RoboDK station: kr30 cnc 041719 works.rdk

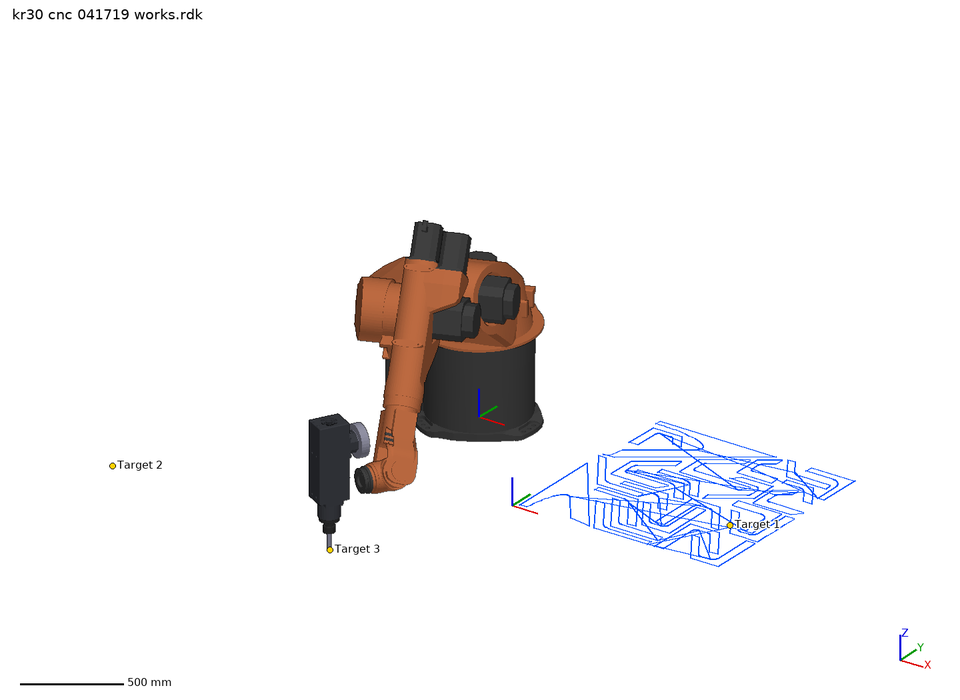
[picture v0: the station drawn from its stored meshes, robots at their saved joint values, targets as dots, program paths as lines]
Station kr30 cnc 041719 works. Poses are relative to the parent item; angles as X-Y-Z fixed-axis rotations.
  - frame KUKA KR 30 HA Base at (0, 0, 0) mm
    - robot KUKA KR 30 HA: 6 axes, payload 30 kg, reach 2033 mm, repeatability 0.05 mm, weight 665 kg
        modified DH rows (alpha deg, a mm, theta deg, d mm): 0, 0, 0, 815; -90, 350, 0, 0; 0, 850, -90, 0; -90, 145, 0, 820; 90, 0, 0, 0; -90, 0, 180, 170
        joint limits [-185, -135, -120, -350, -119, -350] to [185, 35, 158, 350, 119, 350]; home [0, -90, 90, 0, 0, 0]; saved at [68.71, -19.11, 71.06, -56.39, -66.58, 30.88]
      - tool 1/2" End Mill TCP, TCP at (337.71, -2.2, 160.57) mm, size 692.9 x 170 x 256 mm
    - frame Reference Rhino at (909.29, -1020.53, 189.15) mm
      - object RhinoPart at (0, 0, 0) mm
      - target Target 1 (Cartesian target) at (994.45, 406.4, 10) mm, rotated rx 0 ry 90 rz -60.43 deg; joints [10.582, -19.112, 71.071, -56.398, -66.586, 30.882] of KUKA KR 30 HA
      - target Target 2 (Cartesian target) at (-1810.84, -765.32, 10.08) mm, rotated rx 49.23 ry 89.99 rz -110.09 deg; joints [109.49, -19.11, 71.06, -56.39, -66.58, 30.88] of KUKA KR 30 HA
      - target Target 3 (Cartesian target) at (-425.52, -920.6, 10.08) mm, rotated rx 49.23 ry 89.99 rz -69.31 deg; joints [68.71, -19.11, 71.06, -56.39, -66.58, 30.88] of KUKA KR 30 HA
  - machining project RhinoPart Settings: C:/Users/Julian Ramirez.DESKTOP-JVDE542/Desktop/ELMER SHEET 1 TEST 3.nc | rotZ(0) | rotX(00)*rotY(360) | rotZ(0)*rotY(270)
  - object box at (500, 500, 500) mm, size 250 x 250 x 250 mm, geometry from box.sld
  - program RhinoPart (703 instructions, listed below)
  - program Prog2 (1 instructions, listed below)
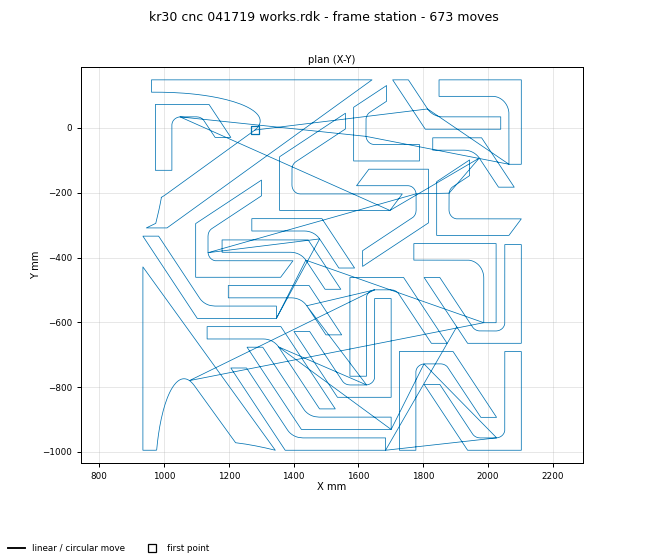
[picture p0: tool path of kr30 cnc 041719 works.rdk in frame station, 673 of 674 moves have a stored position in this frame; points joined in program order, loops and branches not executed]

--- program RhinoPart (robot KUKA KR 30 HA) ---
  Smooth(1)
  Set Ref.: Reference Rhino
  Set Tool: 1/2" End Mill TCP
  Show 1/2" End Mill TCP
  Set speed (2000.0 mm/s)
  MoveJ 1 to (371.32, 1014.09, 0) mm, rotated rx 0 ry 90 rz -60.43 deg; joints [-14.148, -38.783, 129.007, -74.576, -90.059, -0.215]
  MoveL 2 to (371.32, 1014.09, 0) mm, rotated rx 0 ry 90 rz -60.43 deg; joints [-14.148, -38.783, 129.007, -74.576, -90.059, -0.215]
  MoveL 3 to (371.32, 1014.09, 0) mm, rotated rx 0 ry 90 rz -60.43 deg; joints [-14.148, -38.783, 129.007, -74.576, -90.059, -0.215]
  Set speed (60.0 mm/s)
  MoveL 4 to (375.76, 1018.13, 0) mm, rotated rx 0 ry 90 rz -60.43 deg; joints [-14.288, -38.713, 128.612, -74.716, -89.973, 0.097]
  MoveL 5 to (379.48, 1022.21, 0) mm, rotated rx 0 ry 90 rz -60.43 deg; joints [-14.437, -38.65, 128.267, -74.866, -89.9, 0.369]
  MoveL 6 to (382.49, 1026.31, 0) mm, rotated rx 0 ry 90 rz -60.43 deg; joints [-14.595, -38.595, 127.972, -75.024, -89.839, 0.602]
  MoveL 7 to (384.79, 1030.42, 0) mm, rotated rx 0 ry 90 rz -60.43 deg; joints [-14.761, -38.548, 127.726, -75.191, -89.79, 0.795]
  MoveL 8 to (386.4, 1034.54, 0) mm, rotated rx 0 ry 90 rz -60.43 deg; joints [-14.936, -38.511, 127.53, -75.366, -89.752, 0.949]
  MoveL 9 to (387.31, 1038.67, 0) mm, rotated rx 0 ry 90 rz -60.43 deg; joints [-15.118, -38.482, 127.383, -75.549, -89.726, 1.064]
  MoveL 10 to (387.53, 1042.79, 0) mm, rotated rx 0 ry 90 rz -60.43 deg; joints [-15.309, -38.463, 127.286, -75.741, -89.71, 1.141]
  MoveL 11 to (387.07, 1046.9, 0) mm, rotated rx 0 ry 90 rz -60.43 deg; joints [-15.508, -38.454, 127.237, -75.939, -89.704, 1.18]
  MoveL 12 to (385.93, 1051, 0) mm, rotated rx 0 ry 90 rz -60.43 deg; joints [-15.715, -38.454, 127.237, -76.146, -89.709, 1.181]
  MoveL 13 to (384.11, 1055.07, 0) mm, rotated rx 0 ry 90 rz -60.43 deg; joints [-15.929, -38.463, 127.285, -76.36, -89.722, 1.145]
  MoveL 14 to (381.63, 1059.1, 0) mm, rotated rx 0 ry 90 rz -60.43 deg; joints [-16.152, -38.482, 127.38, -76.582, -89.744, 1.071]
  MoveL 15 to (378.49, 1063.11, 0) mm, rotated rx 0 ry 90 rz -60.43 deg; joints [-16.382, -38.509, 127.523, -76.812, -89.775, 0.96]
  MoveL 16 to (374.68, 1067.06, 0) mm, rotated rx 0 ry 90 rz -60.43 deg; joints [-16.62, -38.546, 127.713, -77.05, -89.813, 0.812]
  MoveL 17 to (370.23, 1070.97, 0) mm, rotated rx 0 ry 90 rz -60.43 deg; joints [-16.866, -38.59, 127.949, -77.295, -89.859, 0.626]
  MoveL 18 to (365.13, 1074.81, 0) mm, rotated rx 0 ry 90 rz -60.43 deg; joints [-17.12, -38.643, 128.23, -77.548, -89.911, 0.403]
  MoveL 19 to (356.11, 1080.56, 0) mm, rotated rx 0 ry 90 rz -60.43 deg; joints [-17.523, -38.737, 128.745, -77.951, -90.002, -0.008]
  MoveL 20 to (346.45, 1085.73, 0) mm, rotated rx 0 ry 90 rz -60.43 deg; joints [-17.913, -38.837, 129.313, -78.342, -90.096, -0.467]
  MoveL 21 to (336.49, 1090.32, 0) mm, rotated rx 0 ry 90 rz -60.43 deg; joints [-18.286, -38.938, 129.909, -78.716, -90.19, -0.953]
  MoveL 22 to (326.6, 1094.34, 0) mm, rotated rx 0 ry 90 rz -60.43 deg; joints [-18.636, -39.034, 130.507, -79.068, -90.279, -1.446]
  MoveL 23 to (304.84, 1101.8, 0) mm, rotated rx 0 ry 90 rz -60.43 deg; joints [-19.356, -39.233, 131.838, -79.794, -90.462, -2.563]
  MoveL 24 to (282.07, 1108.12, 0) mm, rotated rx 0 ry 90 rz -60.43 deg; joints [-20.061, -39.416, 133.239, -80.511, -90.631, -3.77]
  MoveL 25 to (259.04, 1113.38, 0) mm, rotated rx 0 ry 90 rz -60.43 deg; joints [-20.745, -39.572, 134.659, -81.207, -90.78, -5.027]
  MoveL 26 to (236.49, 1117.66, 0) mm, rotated rx 0 ry 90 rz -60.43 deg; joints [-21.394, -39.693, 136.047, -81.872, -90.902, -6.29]
  MoveL 27 to (215.72, 1120.95, 0) mm, rotated rx 0 ry 90 rz -60.43 deg; joints [-21.981, -39.774, 137.321, -82.474, -90.994, -7.481]
  MoveL 28 to (194.75, 1123.72, 0) mm, rotated rx 0 ry 90 rz -60.43 deg; joints [-22.566, -39.826, 138.602, -83.075, -91.066, -8.712]
  MoveL 29 to (173.72, 1126.01, 0) mm, rotated rx 0 ry 90 rz -60.43 deg; joints [-23.147, -39.843, 139.881, -83.673, -91.117, -9.976]
  MoveL 30 to (152.78, 1127.82, 0) mm, rotated rx 0 ry 90 rz -60.43 deg; joints [-23.724, -39.824, 141.147, -84.265, -91.146, -11.265]
  MoveL 31 to (132.99, 1129.14, 0) mm, rotated rx 0 ry 90 rz -60.43 deg; joints [-24.268, -39.771, 142.336, -84.822, -91.152, -12.513]
  MoveL 32 to (116.9, 1129.95, 0) mm, rotated rx 0 ry 90 rz -60.43 deg; joints [-24.71, -39.701, 143.298, -85.274, -91.142, -13.55]
  MoveL 33 to (100.77, 1130.52, 0) mm, rotated rx 0 ry 90 rz -60.43 deg; joints [-25.154, -39.606, 144.257, -85.725, -91.116, -14.609]
  MoveL 34 to (84.64, 1130.87, 0) mm, rotated rx 0 ry 90 rz -60.43 deg; joints [-25.598, -39.482, 145.211, -86.175, -91.076, -15.692]
  MoveL 35 to (68.52, 1130.98, 0) mm, rotated rx 0 ry 90 rz -60.43 deg; joints [-26.044, -39.331, 146.159, -86.623, -91.021, -16.798]
  MoveL 36 to (51.93, 1130.98, 0) mm, rotated rx 0 ry 90 rz -60.43 deg; joints [-26.511, -39.143, 147.126, -87.088, -90.945, -17.959]
  MoveL 37 to (51.93, 1169.08, 0) mm, rotated rx 0 ry 90 rz -60.43 deg; joints [-28.654, -39.362, 145.978, -89.121, -90.262, -16.614]
  MoveL 38 to (732.85, 1169.08, 0) mm, rotated rx 0 ry 90 rz -60.43 deg; joints [-16.446, -29.001, 96.264, -77.863, -84.965, 22.201]
  MoveL 39 to (99.83, 711.88, 0) mm, rotated rx 0 ry 90 rz -60.43 deg; joints [1.355, -38.347, 150.049, -60.898, -100.955, -18.85]
  MoveL 40 to (36.02, 711.88, 0) mm, rotated rx 0 ry 90 rz -60.43 deg; joints [1.465, -36.599, 153.958, -61.879, -103.707, -23.912]
  MoveL 41 to (65.11, 725.98, 0) mm, rotated rx 0 ry 90 rz -60.43 deg; joints [0.419, -37.491, 152.214, -62.335, -102.067, -21.741]
  MoveL 42 to (69.92, 745.6, 0) mm, rotated rx 0 ry 90 rz -60.43 deg; joints [-0.957, -37.626, 151.913, -63.561, -101.361, -21.61]
  MoveL 43 to (74.45, 765.38, 0) mm, rotated rx 0 ry 90 rz -60.43 deg; joints [-2.329, -37.76, 151.6, -64.782, -100.662, -21.448]
  MoveL 44 to (78.62, 785.23, 0) mm, rotated rx 0 ry 90 rz -60.43 deg; joints [-3.689, -37.892, 151.279, -65.995, -99.978, -21.26]
  MoveL 45 to (82.38, 805.12, 0) mm, rotated rx 0 ry 90 rz -60.43 deg; joints [-5.036, -38.021, 150.952, -67.198, -99.311, -21.05]
  MoveL 46 to (81.84, 806.04, 0) mm, rotated rx 0 ry 90 rz -60.43 deg; joints [-5.103, -38.01, 150.981, -67.267, -99.302, -21.097]
  MoveL 47 to (85.5, 808.13, 0) mm, rotated rx 0 ry 90 rz -60.43 deg; joints [-5.223, -38.1, 150.742, -67.332, -99.132, -20.808]
  MoveL 48 to (89.1, 810.32, 0) mm, rotated rx 0 ry 90 rz -60.43 deg; joints [-5.349, -38.187, 150.506, -67.404, -98.964, -20.525]
  MoveL 49 to (92.62, 812.61, 0) mm, rotated rx 0 ry 90 rz -60.43 deg; joints [-5.481, -38.27, 150.274, -67.484, -98.797, -20.25]
  MoveL 50 to (96.07, 815.01, 0) mm, rotated rx 0 ry 90 rz -60.43 deg; joints [-5.621, -38.349, 150.044, -67.572, -98.631, -19.981]
  MoveL 51 to (366.16, 1010.08, 0) mm, rotated rx 0 ry 90 rz -60.43 deg; joints [-14.016, -38.861, 129.451, -74.446, -90.158, -0.569]
  MoveL 52 to (371.32, 1014.09, 0) mm, rotated rx 0 ry 90 rz -60.43 deg; joints [-14.148, -38.783, 129.007, -74.576, -90.059, -0.215]
  MoveL 53 to (904.53, 1079.22, 0) mm, rotated rx 0 ry 90 rz -60.43 deg; joints [-11.868, -22.969, 81.101, -74.832, -80.761, 30.636]
  Set speed (60.0 mm/s)
  MoveL 54 to (845.14, 1169.08, 0) mm, rotated rx 0 ry 90 rz -60.43 deg; joints [-15.343, -24.65, 85.19, -77.55, -83.057, 28.702]
  MoveL 55 to (796.61, 1169.08, 0) mm, rotated rx 0 ry 90 rz -60.43 deg; joints [-15.802, -26.637, 90.145, -77.629, -83.905, 25.83]
  MoveL 56 to (897.33, 1016.68, 0) mm, rotated rx 0 ry 90 rz -60.43 deg; joints [-9.818, -23.849, 83.23, -72.827, -80.088, 29.119]
  MoveL 57 to (1130.3, 1016.68, 0) mm, rotated rx 0 ry 90 rz -60.43 deg; joints [-8.62, -9.728, 50.987, -75.829, -74.407, 46.791]
  MoveL 58 to (1130.3, 1054.78, 0) mm, rotated rx 0 ry 90 rz -60.43 deg; joints [-9.753, -9.185, 49.806, -76.795, -75.087, 47.643]
  MoveL 59 to (951.82, 1054.78, 0) mm, rotated rx 0 ry 90 rz -60.43 deg; joints [-10.754, -20.904, 76.185, -74.352, -79.414, 33.26]
  MoveL 60 to (948.36, 1054.88, 0) mm, rotated rx 0 ry 90 rz -60.43 deg; joints [-10.778, -21.079, 76.597, -74.331, -79.491, 33.032]
  MoveL 61 to (944.91, 1055.18, 0) mm, rotated rx 0 ry 90 rz -60.43 deg; joints [-10.81, -21.25, 77, -74.316, -79.571, 32.809]
  MoveL 62 to (941.49, 1055.67, 0) mm, rotated rx 0 ry 90 rz -60.43 deg; joints [-10.847, -21.416, 77.394, -74.308, -79.653, 32.592]
  MoveL 63 to (938.11, 1056.36, 0) mm, rotated rx 0 ry 90 rz -60.43 deg; joints [-10.891, -21.578, 77.777, -74.307, -79.736, 32.383]
  MoveL 64 to (934.77, 1057.25, 0) mm, rotated rx 0 ry 90 rz -60.43 deg; joints [-10.941, -21.734, 78.148, -74.313, -79.821, 32.181]
  MoveL 65 to (931.48, 1058.34, 0) mm, rotated rx 0 ry 90 rz -60.43 deg; joints [-10.998, -21.885, 78.506, -74.326, -79.907, 31.986]
  MoveL 66 to (928.27, 1059.61, 0) mm, rotated rx 0 ry 90 rz -60.43 deg; joints [-11.06, -22.029, 78.85, -74.346, -79.994, 31.801]
  MoveL 67 to (925.13, 1061.08, 0) mm, rotated rx 0 ry 90 rz -60.43 deg; joints [-11.129, -22.167, 79.179, -74.373, -80.082, 31.624]
  MoveL 68 to (922.08, 1062.74, 0) mm, rotated rx 0 ry 90 rz -60.43 deg; joints [-11.204, -22.298, 79.492, -74.407, -80.17, 31.457]
  MoveL 69 to (919.14, 1064.59, 0) mm, rotated rx 0 ry 90 rz -60.43 deg; joints [-11.284, -22.422, 79.786, -74.448, -80.258, 31.302]
  MoveL 70 to (916.32, 1066.61, 0) mm, rotated rx 0 ry 90 rz -60.43 deg; joints [-11.37, -22.536, 80.061, -74.496, -80.345, 31.158]
  MoveL 71 to (913.65, 1068.81, 0) mm, rotated rx 0 ry 90 rz -60.43 deg; joints [-11.46, -22.642, 80.315, -74.551, -80.431, 31.026]
  MoveL 72 to (911.12, 1071.17, 0) mm, rotated rx 0 ry 90 rz -60.43 deg; joints [-11.556, -22.739, 80.547, -74.612, -80.516, 30.908]
  MoveL 73 to (908.75, 1073.7, 0) mm, rotated rx 0 ry 90 rz -60.43 deg; joints [-11.656, -22.826, 80.756, -74.679, -80.599, 30.803]
  MoveL 74 to (906.55, 1076.38, 0) mm, rotated rx 0 ry 90 rz -60.43 deg; joints [-11.76, -22.903, 80.941, -74.752, -80.681, 30.712]
  MoveL 75 to (904.53, 1079.22, 0) mm, rotated rx 0 ry 90 rz -60.43 deg; joints [-11.868, -22.969, 81.101, -74.832, -80.761, 30.636]
  MoveL 76 to (1155.7, 908.41, 0) mm, rotated rx 0 ry 90 rz -60.43 deg; joints [-5.296, -8.63, 48.604, -73.841, -71.636, 47.397]
  Set speed (60.0 mm/s)
  MoveL 77 to (1155.7, 1062.81, 0) mm, rotated rx 0 ry 90 rz -60.43 deg; joints [-9.86, -6.6, 44.232, -77.66, -74.507, 50.684]
  MoveL 78 to (1155.47, 1068.04, 0) mm, rotated rx 0 ry 90 rz -60.43 deg; joints [-10.014, -6.528, 44.077, -77.784, -74.609, 50.794]
  MoveL 79 to (1154.79, 1073.23, 0) mm, rotated rx 0 ry 90 rz -60.43 deg; joints [-10.169, -6.503, 44.023, -77.893, -74.723, 50.85]
  MoveL 80 to (1153.66, 1078.33, 0) mm, rotated rx 0 ry 90 rz -60.43 deg; joints [-10.323, -6.525, 44.07, -77.987, -74.848, 50.852]
  MoveL 81 to (1152.09, 1083.3, 0) mm, rotated rx 0 ry 90 rz -60.43 deg; joints [-10.477, -6.594, 44.218, -78.067, -74.983, 50.797]
  MoveL 82 to (1150.07, 1088.11, 0) mm, rotated rx 0 ry 90 rz -60.43 deg; joints [-10.628, -6.71, 44.467, -78.131, -75.128, 50.688]
  MoveL 83 to (1147.63, 1092.73, 0) mm, rotated rx 0 ry 90 rz -60.43 deg; joints [-10.776, -6.872, 44.815, -78.18, -75.28, 50.525]
  MoveL 84 to (1144.76, 1097.1, 0) mm, rotated rx 0 ry 90 rz -60.43 deg; joints [-10.919, -7.079, 45.259, -78.214, -75.44, 50.309]
  MoveL 85 to (1141.47, 1101.2, 0) mm, rotated rx 0 ry 90 rz -60.43 deg; joints [-11.058, -7.329, 45.797, -78.233, -75.605, 50.041]
  MoveL 86 to (1137.81, 1104.95, 0) mm, rotated rx 0 ry 90 rz -60.43 deg; joints [-11.189, -7.618, 46.419, -78.237, -75.772, 49.726]
  MoveL 87 to (1133.82, 1108.29, 0) mm, rotated rx 0 ry 90 rz -60.43 deg; joints [-11.309, -7.94, 47.112, -78.226, -75.94, 49.37]
  MoveL 88 to (1129.54, 1111.18, 0) mm, rotated rx 0 ry 90 rz -60.43 deg; joints [-11.419, -8.29, 47.868, -78.201, -76.106, 48.979]
  MoveL 89 to (1125, 1113.61, 0) mm, rotated rx 0 ry 90 rz -60.43 deg; joints [-11.518, -8.664, 48.679, -78.163, -76.269, 48.556]
  MoveL 90 to (1120.24, 1115.55, 0) mm, rotated rx 0 ry 90 rz -60.43 deg; joints [-11.603, -9.06, 49.536, -78.112, -76.428, 48.105]
  MoveL 91 to (1115.28, 1116.96, 0) mm, rotated rx 0 ry 90 rz -60.43 deg; joints [-11.675, -9.473, 50.432, -78.048, -76.581, 47.63]
  MoveL 92 to (1110.15, 1117.83, 0) mm, rotated rx 0 ry 90 rz -60.43 deg; joints [-11.732, -9.899, 51.36, -77.971, -76.727, 47.134]
  MoveL 93 to (1104.9, 1118.13, 0) mm, rotated rx 0 ry 90 rz -60.43 deg; joints [-11.773, -10.337, 52.314, -77.881, -76.865, 46.622]
  MoveL 94 to (939.8, 1118.13, 0) mm, rotated rx 0 ry 90 rz -60.43 deg; joints [-12.888, -20.841, 76.037, -76.175, -80.569, 33.658]
  MoveL 95 to (939.8, 1169.08, 0) mm, rotated rx 0 ry 90 rz -60.43 deg; joints [-14.52, -20.204, 74.544, -77.675, -81.292, 34.719]
  MoveL 96 to (1193.8, 1169.08, 0) mm, rotated rx 0 ry 90 rz -60.43 deg; joints [-12.687, 1.86, 26.402, -81.821, -75.178, 60.673]
  MoveL 97 to (1193.8, 908.41, 0) mm, rotated rx 0 ry 90 rz -60.43 deg; joints [-5.193, -4.605, 39.971, -75.302, -70.33, 52.072]
  MoveL 98 to (1155.7, 908.41, 0) mm, rotated rx 0 ry 90 rz -60.43 deg; joints [-5.296, -8.63, 48.604, -73.841, -71.636, 47.397]
  MoveL 99 to (714.35, 994.58, 0) mm, rotated rx 0 ry 90 rz -60.43 deg; joints [-10.182, -31.026, 101.761, -71.621, -83.712, 18.246]
  Set speed (60.0 mm/s)
  MoveL 100 to (714.24, 997.2, 0) mm, rotated rx 0 ry 90 rz -60.43 deg; joints [-10.282, -31.014, 101.729, -71.719, -83.736, 18.276]
  MoveL 101 to (714.24, 1045.45, 0) mm, rotated rx 0 ry 90 rz -60.43 deg; joints [-12.101, -30.702, 100.864, -73.508, -84.152, 18.99]
  MoveL 102 to (714.44, 1048.91, 0) mm, rotated rx 0 ry 90 rz -60.43 deg; joints [-12.229, -30.671, 100.778, -73.635, -84.179, 19.055]
  MoveL 103 to (715.04, 1052.32, 0) mm, rotated rx 0 ry 90 rz -60.43 deg; joints [-12.352, -30.627, 100.656, -73.76, -84.197, 19.142]
  MoveL 104 to (716.03, 1055.63, 0) mm, rotated rx 0 ry 90 rz -60.43 deg; joints [-12.467, -30.57, 100.5, -73.879, -84.207, 19.249]
  MoveL 105 to (717.39, 1058.8, 0) mm, rotated rx 0 ry 90 rz -60.43 deg; joints [-12.574, -30.502, 100.312, -73.992, -84.209, 19.375]
  MoveL 106 to (719.13, 1061.77, 0) mm, rotated rx 0 ry 90 rz -60.43 deg; joints [-12.67, -30.422, 100.094, -74.096, -84.203, 19.518]
  MoveL 107 to (721.23, 1064.5, 0) mm, rotated rx 0 ry 90 rz -60.43 deg; joints [-12.754, -30.332, 99.846, -74.191, -84.188, 19.678]
  MoveL 108 to (723.67, 1066.96, 0) mm, rotated rx 0 ry 90 rz -60.43 deg; joints [-12.824, -30.231, 99.571, -74.275, -84.165, 19.853]
  MoveL 109 to (726.46, 1069.09, 0) mm, rotated rx 0 ry 90 rz -60.43 deg; joints [-12.88, -30.121, 99.271, -74.346, -84.132, 20.043]
  MoveL 110 to (777.74, 1102.98, 0) mm, rotated rx 0 ry 90 rz -60.43 deg; joints [-13.668, -28.021, 93.695, -75.446, -83.519, 23.498]
  MoveL 111 to (777.74, 1151.51, 0) mm, rotated rx 0 ry 90 rz -60.43 deg; joints [-15.376, -27.55, 92.477, -77.095, -84.035, 24.398]
  MoveL 112 to (676.14, 1084.36, 0) mm, rotated rx 0 ry 90 rz -60.43 deg; joints [-13.899, -31.631, 103.464, -75.073, -85.169, 17.533]
  MoveL 113 to (676.14, 918.58, 0) mm, rotated rx 0 ry 90 rz -60.43 deg; joints [-7.466, -32.586, 106.219, -68.709, -83.913, 15.221]
  MoveL 114 to (879.34, 918.58, 0) mm, rotated rx 0 ry 90 rz -60.43 deg; joints [-6.543, -25.264, 86.704, -69.527, -79.221, 26.607]
  MoveL 115 to (879.34, 969.54, 0) mm, rotated rx 0 ry 90 rz -60.43 deg; joints [-8.307, -24.977, 85.996, -71.199, -79.879, 27.302]
  MoveL 116 to (739.64, 969.54, 0) mm, rotated rx 0 ry 90 rz -60.43 deg; joints [-9.074, -30.328, 99.837, -70.701, -82.959, 19.293]
  MoveL 117 to (737.01, 969.69, 0) mm, rotated rx 0 ry 90 rz -60.43 deg; joints [-9.096, -30.416, 100.077, -70.704, -83.016, 19.151]
  MoveL 118 to (734.45, 970.12, 0) mm, rotated rx 0 ry 90 rz -60.43 deg; joints [-9.127, -30.5, 100.307, -70.717, -83.075, 19.015]
  MoveL 119 to (731.97, 970.83, 0) mm, rotated rx 0 ry 90 rz -60.43 deg; joints [-9.169, -30.579, 100.524, -70.741, -83.134, 18.889]
  MoveL 120 to (729.59, 971.8, 0) mm, rotated rx 0 ry 90 rz -60.43 deg; joints [-9.22, -30.653, 100.728, -70.775, -83.193, 18.771]
  MoveL 121 to (727.32, 973.01, 0) mm, rotated rx 0 ry 90 rz -60.43 deg; joints [-9.28, -30.722, 100.918, -70.819, -83.252, 18.662]
  MoveL 122 to (725.18, 974.46, 0) mm, rotated rx 0 ry 90 rz -60.43 deg; joints [-9.348, -30.785, 101.092, -70.871, -83.311, 18.564]
  MoveL 123 to (723.19, 976.13, 0) mm, rotated rx 0 ry 90 rz -60.43 deg; joints [-9.424, -30.841, 101.249, -70.932, -83.367, 18.477]
  MoveL 124 to (721.35, 978, 0) mm, rotated rx 0 ry 90 rz -60.43 deg; joints [-9.507, -30.891, 101.387, -71.002, -83.422, 18.402]
  MoveL 125 to (719.71, 980.05, 0) mm, rotated rx 0 ry 90 rz -60.43 deg; joints [-9.595, -30.934, 101.505, -71.078, -83.475, 18.34]
  MoveL 126 to (718.27, 982.24, 0) mm, rotated rx 0 ry 90 rz -60.43 deg; joints [-9.687, -30.968, 101.602, -71.159, -83.524, 18.291]
  MoveL 127 to (717.05, 984.54, 0) mm, rotated rx 0 ry 90 rz -60.43 deg; joints [-9.783, -30.995, 101.677, -71.245, -83.569, 18.255]
  MoveL 128 to (716.05, 986.95, 0) mm, rotated rx 0 ry 90 rz -60.43 deg; joints [-9.881, -31.015, 101.73, -71.335, -83.611, 18.233]
  MoveL 129 to (715.26, 989.44, 0) mm, rotated rx 0 ry 90 rz -60.43 deg; joints [-9.98, -31.026, 101.762, -71.428, -83.649, 18.224]
  MoveL 130 to (714.69, 991.99, 0) mm, rotated rx 0 ry 90 rz -60.43 deg; joints [-10.081, -31.03, 101.773, -71.524, -83.682, 18.229]
  MoveL 131 to (714.35, 994.58, 0) mm, rotated rx 0 ry 90 rz -60.43 deg; joints [-10.182, -31.026, 101.761, -71.621, -83.712, 18.246]
  MoveL 132 to (139.93, 1054.78, 0) mm, rotated rx 0 ry 90 rz -60.43 deg; joints [-19.98, -39.656, 143.784, -80.693, -92.331, -13.939]
  Set speed (60.0 mm/s)
  MoveL 133 to (137.34, 1054.44, 0) mm, rotated rx 0 ry 90 rz -60.43 deg; joints [-20.014, -39.639, 143.955, -80.734, -92.353, -14.125]
  MoveL 134 to (134.79, 1053.88, 0) mm, rotated rx 0 ry 90 rz -60.43 deg; joints [-20.035, -39.62, 144.127, -80.762, -92.378, -14.314]
  MoveL 135 to (132.3, 1053.09, 0) mm, rotated rx 0 ry 90 rz -60.43 deg; joints [-20.042, -39.601, 144.3, -80.777, -92.408, -14.505]
  MoveL 136 to (129.9, 1052.08, 0) mm, rotated rx 0 ry 90 rz -60.43 deg; joints [-20.035, -39.58, 144.473, -80.778, -92.44, -14.695]
  MoveL 137 to (127.59, 1050.86, 0) mm, rotated rx 0 ry 90 rz -60.43 deg; joints [-20.013, -39.559, 144.644, -80.765, -92.477, -14.885]
  MoveL 138 to (125.4, 1049.43, 0) mm, rotated rx 0 ry 90 rz -60.43 deg; joints [-19.976, -39.537, 144.812, -80.737, -92.517, -15.071]
  MoveL 139 to (123.35, 1047.78, 0) mm, rotated rx 0 ry 90 rz -60.43 deg; joints [-19.923, -39.515, 144.976, -80.695, -92.561, -15.253]
  MoveL 140 to (121.48, 1045.95, 0) mm, rotated rx 0 ry 90 rz -60.43 deg; joints [-19.856, -39.493, 145.134, -80.638, -92.608, -15.427]
  MoveL 141 to (119.81, 1043.95, 0) mm, rotated rx 0 ry 90 rz -60.43 deg; joints [-19.775, -39.472, 145.282, -80.567, -92.657, -15.59]
  MoveL 142 to (118.36, 1041.82, 0) mm, rotated rx 0 ry 90 rz -60.43 deg; joints [-19.68, -39.452, 145.419, -80.483, -92.709, -15.741]
  MoveL 143 to (117.15, 1039.55, 0) mm, rotated rx 0 ry 90 rz -60.43 deg; joints [-19.572, -39.433, 145.544, -80.386, -92.762, -15.879]
  MoveL 144 to (116.18, 1037.16, 0) mm, rotated rx 0 ry 90 rz -60.43 deg; joints [-19.452, -39.415, 145.656, -80.277, -92.817, -16.001]
  MoveL 145 to (115.47, 1034.68, 0) mm, rotated rx 0 ry 90 rz -60.43 deg; joints [-19.321, -39.399, 145.754, -80.155, -92.872, -16.107]
  MoveL 146 to (115.04, 1032.12, 0) mm, rotated rx 0 ry 90 rz -60.43 deg; joints [-19.178, -39.386, 145.836, -80.023, -92.928, -16.194]
  MoveL 147 to (114.89, 1029.5, 0) mm, rotated rx 0 ry 90 rz -60.43 deg; joints [-19.025, -39.375, 145.901, -79.88, -92.984, -16.262]
  MoveL 148 to (114.89, 889.8, 0) mm, rotated rx 0 ry 90 rz -60.43 deg; joints [-10.367, -38.892, 148.202, -71.802, -96.244, -18.308]
  MoveL 149 to (63.94, 889.8, 0) mm, rotated rx 0 ry 90 rz -60.43 deg; joints [-11.002, -37.862, 151.353, -72.876, -97.292, -22.391]
  MoveL 150 to (63.94, 1093, 0) mm, rotated rx 0 ry 90 rz -60.43 deg; joints [-23.973, -39.068, 147.471, -84.686, -91.765, -18.321]
  MoveL 151 to (229.71, 1093, 0) mm, rotated rx 0 ry 90 rz -60.43 deg; joints [-20.268, -39.763, 137.112, -80.771, -91.185, -7.253]
  MoveL 152 to (296.86, 991.4, 0) mm, rotated rx 0 ry 90 rz -60.43 deg; joints [-13.945, -39.574, 134.678, -74.432, -91.373, -4.916]
  MoveL 153 to (248.33, 991.4, 0) mm, rotated rx 0 ry 90 rz -60.43 deg; joints [-14.596, -39.806, 138, -75.17, -92.111, -7.92]
  MoveL 154 to (214.44, 1042.68, 0) mm, rotated rx 0 ry 90 rz -60.43 deg; joints [-17.893, -39.839, 139.265, -78.474, -91.9, -9.234]
  MoveL 155 to (212.31, 1045.46, 0) mm, rotated rx 0 ry 90 rz -60.43 deg; joints [-18.08, -39.84, 139.345, -78.662, -91.885, -9.318]
  MoveL 156 to (209.86, 1047.91, 0) mm, rotated rx 0 ry 90 rz -60.43 deg; joints [-18.256, -39.841, 139.454, -78.839, -91.878, -9.429]
  MoveL 157 to (207.12, 1050.01, 0) mm, rotated rx 0 ry 90 rz -60.43 deg; joints [-18.418, -39.842, 139.587, -79.003, -91.876, -9.564]
  MoveL 158 to (204.15, 1051.74, 0) mm, rotated rx 0 ry 90 rz -60.43 deg; joints [-18.565, -39.843, 139.744, -79.154, -91.881, -9.722]
  MoveL 159 to (200.98, 1053.11, 0) mm, rotated rx 0 ry 90 rz -60.43 deg; joints [-18.697, -39.843, 139.92, -79.289, -91.892, -9.899]
  MoveL 160 to (197.68, 1054.09, 0) mm, rotated rx 0 ry 90 rz -60.43 deg; joints [-18.811, -39.842, 140.113, -79.408, -91.908, -10.094]
  MoveL 161 to (190.8, 1054.9, 0) mm, rotated rx 0 ry 90 rz -60.43 deg; joints [-18.983, -39.838, 140.542, -79.592, -91.956, -10.526]
  MoveL 162 to (142.55, 1054.9, 0) mm, rotated rx 0 ry 90 rz -60.43 deg; joints [-19.932, -39.672, 143.618, -80.64, -92.313, -13.756]
  MoveL 163 to (139.93, 1054.78, 0) mm, rotated rx 0 ry 90 rz -60.43 deg; joints [-19.98, -39.656, 143.784, -80.693, -92.331, -13.939]
  MoveL 164 to (788.26, 765.88, 0) mm, rotated rx 0 ry 90 rz -60.43 deg; joints [-1.266, -29.269, 96.976, -63.512, -79.638, 19.847]
  Set speed (60.0 mm/s)
  MoveL 165 to (826.36, 816.83, 0) mm, rotated rx 0 ry 90 rz -60.43 deg; joints [-3.087, -27.773, 93.052, -65.649, -79.251, 22.395]
  MoveL 166 to (511.04, 816.83, 0) mm, rotated rx 0 ry 90 rz -60.43 deg; joints [-3.857, -36.982, 120.764, -64.418, -87.306, 5.606]
  MoveL 167 to (505.85, 817.41, 0) mm, rotated rx 0 ry 90 rz -60.43 deg; joints [-3.9, -37.085, 121.169, -64.448, -87.441, 5.336]
  MoveL 168 to (503.37, 818.12, 0) mm, rotated rx 0 ry 90 rz -60.43 deg; joints [-3.94, -37.133, 121.36, -64.482, -87.506, 5.208]
  MoveL 169 to (500.99, 819.09, 0) mm, rotated rx 0 ry 90 rz -60.43 deg; joints [-3.991, -37.178, 121.541, -64.528, -87.569, 5.088]
  MoveL 170 to (498.72, 820.3, 0) mm, rotated rx 0 ry 90 rz -60.43 deg; joints [-4.054, -37.221, 121.712, -64.586, -87.63, 4.974]
  MoveL 171 to (496.58, 821.75, 0) mm, rotated rx 0 ry 90 rz -60.43 deg; joints [-4.127, -37.26, 121.871, -64.654, -87.688, 4.869]
  MoveL 172 to (494.59, 823.42, 0) mm, rotated rx 0 ry 90 rz -60.43 deg; joints [-4.211, -37.296, 122.017, -64.733, -87.742, 4.772]
  MoveL 173 to (492.75, 825.29, 0) mm, rotated rx 0 ry 90 rz -60.43 deg; joints [-4.303, -37.328, 122.149, -64.822, -87.792, 4.686]
  MoveL 174 to (491.11, 827.34, 0) mm, rotated rx 0 ry 90 rz -60.43 deg; joints [-4.403, -37.357, 122.265, -64.918, -87.837, 4.61]
  MoveL 175 to (489.67, 829.53, 0) mm, rotated rx 0 ry 90 rz -60.43 deg; joints [-4.509, -37.381, 122.364, -65.021, -87.877, 4.547]
  MoveL 176 to (487.45, 834.24, 0) mm, rotated rx 0 ry 90 rz -60.43 deg; joints [-4.734, -37.415, 122.507, -65.242, -87.94, 4.456]
  MoveL 177 to (486.09, 839.28, 0) mm, rotated rx 0 ry 90 rz -60.43 deg; joints [-4.971, -37.433, 122.579, -65.477, -87.982, 4.415]
  MoveL 178 to (485.64, 844.49, 0) mm, rotated rx 0 ry 90 rz -60.43 deg; joints [-5.213, -37.432, 122.578, -65.719, -88, 4.424]
  MoveL 179 to (485.64, 892.74, 0) mm, rotated rx 0 ry 90 rz -60.43 deg; joints [-7.426, -37.332, 122.164, -67.936, -88.054, 4.789]
  MoveL 180 to (485.84, 896.21, 0) mm, rotated rx 0 ry 90 rz -60.43 deg; joints [-7.583, -37.319, 122.113, -68.094, -88.053, 4.83]
  MoveL 181 to (486.44, 899.62, 0) mm, rotated rx 0 ry 90 rz -60.43 deg; joints [-7.735, -37.299, 122.031, -68.247, -88.043, 4.892]
  MoveL 182 to (487.43, 902.93, 0) mm, rotated rx 0 ry 90 rz -60.43 deg; joints [-7.88, -37.272, 121.919, -68.394, -88.024, 4.976]
  MoveL 183 to (488.79, 906.09, 0) mm, rotated rx 0 ry 90 rz -60.43 deg; joints [-8.015, -37.237, 121.779, -68.532, -87.997, 5.079]
  MoveL 184 to (490.53, 909.06, 0) mm, rotated rx 0 ry 90 rz -60.43 deg; joints [-8.139, -37.196, 121.611, -68.66, -87.962, 5.2]
  MoveL 185 to (492.63, 911.8, 0) mm, rotated rx 0 ry 90 rz -60.43 deg; joints [-8.249, -37.148, 121.418, -68.774, -87.92, 5.34]
  MoveL 186 to (495.07, 914.25, 0) mm, rotated rx 0 ry 90 rz -60.43 deg; joints [-8.344, -37.093, 121.2, -68.874, -87.87, 5.496]
  MoveL 187 to (497.86, 916.38, 0) mm, rotated rx 0 ry 90 rz -60.43 deg; joints [-8.421, -37.032, 120.958, -68.958, -87.812, 5.667]
  MoveL 188 to (650.74, 1017.42, 0) mm, rotated rx 0 ry 90 rz -60.43 deg; joints [-11.535, -32.847, 106.99, -72.608, -85.147, 15.114]
  MoveL 189 to (650.74, 1065.95, 0) mm, rotated rx 0 ry 90 rz -60.43 deg; joints [-13.43, -32.533, 106.064, -74.488, -85.48, 15.852]
  MoveL 190 to (447.54, 931.66, 0) mm, rotated rx 0 ry 90 rz -60.43 deg; joints [-9.484, -37.91, 124.64, -69.942, -88.877, 3.071]
  MoveL 191 to (447.54, 765.88, 0) mm, rotated rx 0 ry 90 rz -60.43 deg; joints [-1.626, -38.176, 125.869, -62.074, -88.919, 2.038]
  MoveL 192 to (788.26, 765.88, 0) mm, rotated rx 0 ry 90 rz -60.43 deg; joints [-1.266, -29.269, 96.976, -63.512, -79.638, 19.847]
  MoveL 193 to (1064.06, 927.56, 0) mm, rotated rx 0 ry 90 rz -60.43 deg; joints [-6.162, -15.538, 63.842, -72.085, -74.676, 39.266]
  Set speed (60.0 mm/s)
  MoveL 194 to (1062.04, 930.4, 0) mm, rotated rx 0 ry 90 rz -60.43 deg; joints [-6.257, -15.649, 64.092, -72.126, -74.779, 39.149]
  MoveL 195 to (1059.84, 933.08, 0) mm, rotated rx 0 ry 90 rz -60.43 deg; joints [-6.349, -15.772, 64.37, -72.16, -74.884, 39.016]
  MoveL 196 to (1057.47, 935.61, 0) mm, rotated rx 0 ry 90 rz -60.43 deg; joints [-6.436, -15.906, 64.673, -72.187, -74.991, 38.868]
  MoveL 197 to (1054.94, 937.97, 0) mm, rotated rx 0 ry 90 rz -60.43 deg; joints [-6.519, -16.051, 64.999, -72.208, -75.098, 38.706]
  MoveL 198 to (1052.26, 940.17, 0) mm, rotated rx 0 ry 90 rz -60.43 deg; joints [-6.598, -16.204, 65.347, -72.222, -75.207, 38.531]
  MoveL 199 to (1049.45, 942.19, 0) mm, rotated rx 0 ry 90 rz -60.43 deg; joints [-6.672, -16.367, 65.715, -72.231, -75.315, 38.344]
  MoveL 200 to (1046.51, 944.04, 0) mm, rotated rx 0 ry 90 rz -60.43 deg; joints [-6.741, -16.537, 66.1, -72.233, -75.424, 38.146]
  MoveL 201 to (1043.45, 945.7, 0) mm, rotated rx 0 ry 90 rz -60.43 deg; joints [-6.805, -16.714, 66.502, -72.23, -75.532, 37.938]
  MoveL 202 to (1040.31, 947.17, 0) mm, rotated rx 0 ry 90 rz -60.43 deg; joints [-6.863, -16.896, 66.916, -72.22, -75.638, 37.722]
  MoveL 203 to (1037.1, 948.45, 0) mm, rotated rx 0 ry 90 rz -60.43 deg; joints [-6.915, -17.082, 67.341, -72.205, -75.743, 37.499]
  MoveL 204 to (1033.82, 949.53, 0) mm, rotated rx 0 ry 90 rz -60.43 deg; joints [-6.962, -17.273, 67.775, -72.185, -75.846, 37.269]
  MoveL 205 to (1030.48, 950.42, 0) mm, rotated rx 0 ry 90 rz -60.43 deg; joints [-7.003, -17.466, 68.217, -72.16, -75.947, 37.033]
  MoveL 206 to (1027.09, 951.11, 0) mm, rotated rx 0 ry 90 rz -60.43 deg; joints [-7.039, -17.662, 68.665, -72.129, -76.045, 36.793]
  MoveL 207 to (1023.67, 951.61, 0) mm, rotated rx 0 ry 90 rz -60.43 deg; joints [-7.068, -17.86, 69.118, -72.093, -76.141, 36.549]
  MoveL 208 to (1020.23, 951.9, 0) mm, rotated rx 0 ry 90 rz -60.43 deg; joints [-7.091, -18.059, 69.574, -72.052, -76.234, 36.301]
  MoveL 209 to (1016.77, 952, 0) mm, rotated rx 0 ry 90 rz -60.43 deg; joints [-7.108, -18.259, 70.033, -72.006, -76.324, 36.051]
  MoveL 210 to (920.39, 952, 0) mm, rotated rx 0 ry 90 rz -60.43 deg; joints [-7.514, -23.243, 81.76, -70.937, -78.69, 29.577]
  MoveL 211 to (920.39, 990.1, 0) mm, rotated rx 0 ry 90 rz -60.43 deg; joints [-8.796, -22.987, 81.144, -72.137, -79.214, 30.143]
  MoveL 212 to (1071.25, 990.1, 0) mm, rotated rx 0 ry 90 rz -60.43 deg; joints [-8.077, -14.538, 61.598, -73.918, -75.545, 40.888]
  MoveL 213 to (1171.98, 837.7, 0) mm, rotated rx 0 ry 90 rz -60.43 deg; joints [-3.153, -7.564, 46.301, -72.731, -69.693, 48.146]
  MoveL 214 to (1123.45, 837.7, 0) mm, rotated rx 0 ry 90 rz -60.43 deg; joints [-3.235, -11.829, 55.587, -71.101, -71.311, 43.105]
  MoveL 215 to (1064.06, 927.56, 0) mm, rotated rx 0 ry 90 rz -60.43 deg; joints [-6.162, -15.538, 63.842, -72.085, -74.676, 39.266]
  MoveL 216 to (970.82, 819.19, 0) mm, rotated rx 0 ry 90 rz -60.43 deg; joints [-2.906, -21.375, 77.297, -67.415, -75.436, 31.155]
  Set speed (60.0 mm/s)
  MoveL 217 to (971.42, 822.6, 0) mm, rotated rx 0 ry 90 rz -60.43 deg; joints [-3.019, -21.336, 77.204, -67.527, -75.474, 31.231]
  MoveL 218 to (972.4, 825.91, 0) mm, rotated rx 0 ry 90 rz -60.43 deg; joints [-3.127, -21.276, 77.064, -67.642, -75.499, 31.332]
  MoveL 219 to (973.77, 829.08, 0) mm, rotated rx 0 ry 90 rz -60.43 deg; joints [-3.229, -21.198, 76.878, -67.758, -75.512, 31.457]
  MoveL 220 to (975.51, 832.05, 0) mm, rotated rx 0 ry 90 rz -60.43 deg; joints [-3.324, -21.1, 76.647, -67.874, -75.511, 31.605]
  MoveL 221 to (977.6, 834.78, 0) mm, rotated rx 0 ry 90 rz -60.43 deg; joints [-3.411, -20.984, 76.373, -67.988, -75.497, 31.775]
  MoveL 222 to (980.05, 837.24, 0) mm, rotated rx 0 ry 90 rz -60.43 deg; joints [-3.487, -20.849, 76.057, -68.098, -75.47, 31.967]
  MoveL 223 to (982.84, 839.37, 0) mm, rotated rx 0 ry 90 rz -60.43 deg; joints [-3.552, -20.697, 75.699, -68.204, -75.427, 32.178]
  MoveL 224 to (1034.12, 873.26, 0) mm, rotated rx 0 ry 90 rz -60.43 deg; joints [-4.534, -17.714, 68.782, -70.031, -74.577, 36.2]
  MoveL 225 to (1034.12, 921.79, 0) mm, rotated rx 0 ry 90 rz -60.43 deg; joints [-6.081, -17.445, 68.168, -71.405, -75.384, 36.871]
  MoveL 226 to (932.52, 854.64, 0) mm, rotated rx 0 ry 90 rz -60.43 deg; joints [-4.176, -23.142, 81.516, -67.99, -77.004, 29.088]
  MoveL 227 to (932.52, 688.86, 0) mm, rotated rx 0 ry 90 rz -60.43 deg; joints [1.468, -23.326, 81.962, -62.803, -74.432, 27.577]
  MoveL 228 to (1155.67, 688.86, 0) mm, rotated rx 0 ry 90 rz -60.43 deg; joints [1.296, -9.337, 50.136, -68.666, -67.146, 44.84]
  MoveL 229 to (1193.77, 739.82, 0) mm, rotated rx 0 ry 90 rz -60.43 deg; joints [-0.233, -5.55, 41.984, -71.54, -66.784, 49.742]
  MoveL 230 to (996.02, 739.82, 0) mm, rotated rx 0 ry 90 rz -60.43 deg; joints [-0.259, -20.175, 74.476, -65.489, -73.4, 32.07]
  MoveL 231 to (993.39, 739.97, 0) mm, rotated rx 0 ry 90 rz -60.43 deg; joints [-0.264, -20.315, 74.804, -65.443, -73.481, 31.893]
  MoveL 232 to (990.83, 740.4, 0) mm, rotated rx 0 ry 90 rz -60.43 deg; joints [-0.279, -20.451, 75.121, -65.407, -73.565, 31.724]
  MoveL 233 to (988.35, 741.11, 0) mm, rotated rx 0 ry 90 rz -60.43 deg; joints [-0.303, -20.582, 75.428, -65.381, -73.65, 31.563]
  MoveL 234 to (985.96, 742.08, 0) mm, rotated rx 0 ry 90 rz -60.43 deg; joints [-0.335, -20.706, 75.721, -65.365, -73.737, 31.412]
  MoveL 235 to (983.7, 743.29, 0) mm, rotated rx 0 ry 90 rz -60.43 deg; joints [-0.376, -20.824, 75.998, -65.359, -73.825, 31.271]
  MoveL 236 to (981.56, 744.74, 0) mm, rotated rx 0 ry 90 rz -60.43 deg; joints [-0.424, -20.935, 76.258, -65.363, -73.912, 31.141]
  MoveL 237 to (979.56, 746.41, 0) mm, rotated rx 0 ry 90 rz -60.43 deg; joints [-0.48, -21.037, 76.5, -65.376, -73.999, 31.024]
  MoveL 238 to (977.73, 748.28, 0) mm, rotated rx 0 ry 90 rz -60.43 deg; joints [-0.543, -21.131, 76.72, -65.399, -74.084, 30.919]
  MoveL 239 to (976.08, 750.33, 0) mm, rotated rx 0 ry 90 rz -60.43 deg; joints [-0.611, -21.214, 76.917, -65.431, -74.167, 30.829]
  MoveL 240 to (974.65, 752.52, 0) mm, rotated rx 0 ry 90 rz -60.43 deg; joints [-0.685, -21.286, 77.087, -65.471, -74.245, 30.753]
  MoveL 241 to (973.43, 754.82, 0) mm, rotated rx 0 ry 90 rz -60.43 deg; joints [-0.762, -21.347, 77.231, -65.519, -74.319, 30.694]
  MoveL 242 to (972.42, 757.23, 0) mm, rotated rx 0 ry 90 rz -60.43 deg; joints [-0.842, -21.397, 77.348, -65.574, -74.388, 30.649]
  MoveL 243 to (971.64, 759.72, 0) mm, rotated rx 0 ry 90 rz -60.43 deg; joints [-0.926, -21.435, 77.438, -65.635, -74.452, 30.62]
  MoveL 244 to (971.07, 762.27, 0) mm, rotated rx 0 ry 90 rz -60.43 deg; joints [-1.011, -21.461, 77.501, -65.702, -74.51, 30.606]
  MoveL 245 to (970.73, 764.86, 0) mm, rotated rx 0 ry 90 rz -60.43 deg; joints [-1.097, -21.476, 77.536, -65.774, -74.562, 30.608]
  MoveL 246 to (970.62, 767.48, 0) mm, rotated rx 0 ry 90 rz -60.43 deg; joints [-1.185, -21.479, 77.543, -65.851, -74.609, 30.624]
  MoveL 247 to (970.62, 815.73, 0) mm, rotated rx 0 ry 90 rz -60.43 deg; joints [-2.791, -21.394, 77.342, -67.307, -75.387, 31.104]
  MoveL 248 to (970.82, 819.19, 0) mm, rotated rx 0 ry 90 rz -60.43 deg; joints [-2.906, -21.375, 77.297, -67.415, -75.436, 31.155]
  MoveL 249 to (868.9, 817.19, 0) mm, rotated rx 0 ry 90 rz -60.43 deg; joints [-3.018, -26.065, 88.703, -66.067, -78.144, 24.84]
  Set speed (60.0 mm/s)
  MoveL 250 to (868.56, 819.78, 0) mm, rotated rx 0 ry 90 rz -60.43 deg; joints [-3.111, -26.073, 88.724, -66.15, -78.188, 24.846]
  MoveL 251 to (867.99, 822.33, 0) mm, rotated rx 0 ry 90 rz -60.43 deg; joints [-3.202, -26.091, 88.768, -66.229, -78.237, 24.838]
  MoveL 252 to (867.21, 824.82, 0) mm, rotated rx 0 ry 90 rz -60.43 deg; joints [-3.291, -26.118, 88.836, -66.305, -78.291, 24.817]
  MoveL 253 to (866.2, 827.22, 0) mm, rotated rx 0 ry 90 rz -60.43 deg; joints [-3.378, -26.154, 88.926, -66.375, -78.349, 24.783]
  MoveL 254 to (864.98, 829.53, 0) mm, rotated rx 0 ry 90 rz -60.43 deg; joints [-3.462, -26.199, 89.039, -66.44, -78.411, 24.735]
  MoveL 255 to (863.55, 831.72, 0) mm, rotated rx 0 ry 90 rz -60.43 deg; joints [-3.543, -26.252, 89.175, -66.5, -78.478, 24.673]
  MoveL 256 to (861.9, 833.77, 0) mm, rotated rx 0 ry 90 rz -60.43 deg; joints [-3.619, -26.315, 89.332, -66.553, -78.547, 24.598]
  MoveL 257 to (860.07, 835.64, 0) mm, rotated rx 0 ry 90 rz -60.43 deg; joints [-3.69, -26.385, 89.51, -66.598, -78.619, 24.511]
  MoveL 258 to (858.07, 837.31, 0) mm, rotated rx 0 ry 90 rz -60.43 deg; joints [-3.754, -26.463, 89.705, -66.636, -78.693, 24.412]
  MoveL 259 to (855.93, 838.76, 0) mm, rotated rx 0 ry 90 rz -60.43 deg; joints [-3.81, -26.546, 89.916, -66.665, -78.766, 24.303]
  MoveL 260 to (853.67, 839.97, 0) mm, rotated rx 0 ry 90 rz -60.43 deg; joints [-3.859, -26.635, 90.142, -66.685, -78.84, 24.184]
  MoveL 261 to (851.28, 840.94, 0) mm, rotated rx 0 ry 90 rz -60.43 deg; joints [-3.899, -26.729, 90.38, -66.697, -78.914, 24.057]
  MoveL 262 to (848.8, 841.65, 0) mm, rotated rx 0 ry 90 rz -60.43 deg; joints [-3.93, -26.827, 90.629, -66.699, -78.986, 23.921]
  MoveL 263 to (846.24, 842.08, 0) mm, rotated rx 0 ry 90 rz -60.43 deg; joints [-3.952, -26.929, 90.888, -66.691, -79.057, 23.778]
  MoveL 264 to (843.62, 842.23, 0) mm, rotated rx 0 ry 90 rz -60.43 deg; joints [-3.964, -27.034, 91.155, -66.674, -79.126, 23.628]
  MoveL 265 to (685.05, 842.23, 0) mm, rotated rx 0 ry 90 rz -60.43 deg; joints [-4.401, -32.557, 106.134, -65.736, -83.094, 14.936]
  MoveL 266 to (723.15, 893.18, 0) mm, rotated rx 0 ry 90 rz -60.43 deg; joints [-6.255, -31.216, 102.293, -67.818, -82.625, 17.475]
  MoveL 267 to (907.12, 893.18, 0) mm, rotated rx 0 ry 90 rz -60.43 deg; joints [-5.564, -24.161, 83.99, -68.941, -78.201, 27.97]
  MoveL 268 to (907.12, 727.4, 0) mm, rotated rx 0 ry 90 rz -60.43 deg; joints [0.157, -24.512, 84.851, -63.609, -75.794, 26.314]
  MoveL 269 to (703.92, 593.11, 0) mm, rotated rx 0 ry 90 rz -60.43 deg; joints [5.462, -31.902, 104.237, -56.257, -79.968, 14.615]
  MoveL 270 to (703.92, 641.64, 0) mm, rotated rx 0 ry 90 rz -60.43 deg; joints [3.558, -32.021, 104.58, -58.092, -80.572, 14.74]
  MoveL 271 to (856.79, 742.68, 0) mm, rotated rx 0 ry 90 rz -60.43 deg; joints [-0.384, -26.655, 90.191, -63.432, -77.448, 23.489]
  MoveL 272 to (859.58, 744.81, 0) mm, rotated rx 0 ry 90 rz -60.43 deg; joints [-0.459, -26.54, 89.901, -63.537, -77.4, 23.665]
  MoveL 273 to (862.03, 747.26, 0) mm, rotated rx 0 ry 90 rz -60.43 deg; joints [-0.546, -26.439, 89.646, -63.65, -77.366, 23.825]
  MoveL 274 to (864.12, 750, 0) mm, rotated rx 0 ry 90 rz -60.43 deg; joints [-0.642, -26.352, 89.425, -63.767, -77.346, 23.967]
  MoveL 275 to (865.86, 752.97, 0) mm, rotated rx 0 ry 90 rz -60.43 deg; joints [-0.747, -26.279, 89.241, -63.887, -77.34, 24.091]
  MoveL 276 to (867.23, 756.13, 0) mm, rotated rx 0 ry 90 rz -60.43 deg; joints [-0.858, -26.22, 89.094, -64.009, -77.347, 24.195]
  MoveL 277 to (868.21, 759.44, 0) mm, rotated rx 0 ry 90 rz -60.43 deg; joints [-0.975, -26.177, 88.985, -64.132, -77.366, 24.279]
  MoveL 278 to (869.02, 766.32, 0) mm, rotated rx 0 ry 90 rz -60.43 deg; joints [-1.218, -26.138, 88.888, -64.371, -77.441, 24.383]
  MoveL 279 to (869.02, 814.57, 0) mm, rotated rx 0 ry 90 rz -60.43 deg; joints [-2.926, -26.066, 88.705, -65.98, -78.105, 24.821]
  MoveL 280 to (868.9, 817.19, 0) mm, rotated rx 0 ry 90 rz -60.43 deg; joints [-3.018, -26.065, 88.703, -66.067, -78.144, 24.84]
  MoveL 281 to (226.56, 635.47, 0) mm, rotated rx 0 ry 90 rz -60.43 deg; joints [5.652, -39.814, 141.461, -55.336, -96.687, -9.558]
  Set speed (60.0 mm/s)
  MoveL 282 to (226.44, 638.09, 0) mm, rotated rx 0 ry 90 rz -60.43 deg; joints [5.5, -39.813, 141.486, -55.489, -96.676, -9.597]
  MoveL 283 to (226.44, 686.34, 0) mm, rotated rx 0 ry 90 rz -60.43 deg; joints [2.678, -39.803, 141.719, -58.311, -96.326, -10.119]
  MoveL 284 to (227.25, 693.22, 0) mm, rotated rx 0 ry 90 rz -60.43 deg; joints [2.273, -39.805, 141.685, -58.709, -96.236, -10.132]
  MoveL 285 to (228.23, 696.53, 0) mm, rotated rx 0 ry 90 rz -60.43 deg; joints [2.077, -39.807, 141.627, -58.897, -96.17, -10.101]
  MoveL 286 to (229.6, 699.69, 0) mm, rotated rx 0 ry 90 rz -60.43 deg; joints [1.889, -39.811, 141.541, -59.076, -96.091, -10.044]
  MoveL 287 to (231.33, 702.66, 0) mm, rotated rx 0 ry 90 rz -60.43 deg; joints [1.712, -39.815, 141.43, -59.24, -96.001, -9.963]
  MoveL 288 to (233.43, 705.4, 0) mm, rotated rx 0 ry 90 rz -60.43 deg; joints [1.548, -39.82, 141.293, -59.389, -95.9, -9.857]
  MoveL 289 to (235.88, 707.86, 0) mm, rotated rx 0 ry 90 rz -60.43 deg; joints [1.402, -39.825, 141.131, -59.52, -95.791, -9.727]
  MoveL 290 to (238.67, 709.99, 0) mm, rotated rx 0 ry 90 rz -60.43 deg; joints [1.274, -39.83, 140.944, -59.63, -95.672, -9.573]
  MoveL 291 to (391.54, 811.03, 0) mm, rotated rx 0 ry 90 rz -60.43 deg; joints [-3.97, -38.936, 129.9, -64.402, -90.417, -0.87]
  MoveL 292 to (391.54, 859.56, 0) mm, rotated rx 0 ry 90 rz -60.43 deg; joints [-6.39, -38.882, 129.576, -66.82, -90.273, -0.638]
  MoveL 293 to (188.34, 725.26, 0) mm, rotated rx 0 ry 90 rz -60.43 deg; joints [0.408, -39.595, 144.345, -60.844, -97.309, -12.846]
  MoveL 294 to (188.34, 559.48, 0) mm, rotated rx 0 ry 90 rz -60.43 deg; joints [10.435, -39.701, 143.297, -50.793, -98.692, -10.495]
  MoveL 295 to (450.69, 559.48, 0) mm, rotated rx 0 ry 90 rz -60.43 deg; joints [8.186, -37.928, 124.722, -52.285, -88.038, 2.535]
  MoveL 296 to (488.79, 610.43, 0) mm, rotated rx 0 ry 90 rz -60.43 deg; joints [5.61, -37.357, 122.268, -54.925, -87.07, 4.163]
  MoveL 297 to (251.84, 610.43, 0) mm, rotated rx 0 ry 90 rz -60.43 deg; joints [6.928, -39.842, 139.552, -53.895, -95.758, -7.832]
  MoveL 298 to (249.22, 610.58, 0) mm, rotated rx 0 ry 90 rz -60.43 deg; joints [6.938, -39.843, 139.733, -53.9, -95.865, -7.977]
  MoveL 299 to (246.66, 611.02, 0) mm, rotated rx 0 ry 90 rz -60.43 deg; joints [6.931, -39.843, 139.911, -53.922, -95.969, -8.123]
  MoveL 300 to (244.18, 611.72, 0) mm, rotated rx 0 ry 90 rz -60.43 deg; joints [6.908, -39.842, 140.087, -53.96, -96.069, -8.268]
  MoveL 301 to (241.79, 612.69, 0) mm, rotated rx 0 ry 90 rz -60.43 deg; joints [6.869, -39.841, 140.257, -54.013, -96.165, -8.412]
  MoveL 302 to (239.53, 613.91, 0) mm, rotated rx 0 ry 90 rz -60.43 deg; joints [6.815, -39.84, 140.421, -54.081, -96.254, -8.553]
  MoveL 303 to (237.39, 615.35, 0) mm, rotated rx 0 ry 90 rz -60.43 deg; joints [6.747, -39.837, 140.578, -54.164, -96.337, -8.69]
  MoveL 304 to (235.39, 617.02, 0) mm, rotated rx 0 ry 90 rz -60.43 deg; joints [6.664, -39.835, 140.727, -54.259, -96.413, -8.823]
  MoveL 305 to (233.56, 618.9, 0) mm, rotated rx 0 ry 90 rz -60.43 deg; joints [6.569, -39.832, 140.866, -54.367, -96.481, -8.95]
  MoveL 306 to (231.91, 620.95, 0) mm, rotated rx 0 ry 90 rz -60.43 deg; joints [6.461, -39.829, 140.994, -54.486, -96.541, -9.069]
  MoveL 307 to (230.48, 623.13, 0) mm, rotated rx 0 ry 90 rz -60.43 deg; joints [6.344, -39.826, 141.108, -54.614, -96.59, -9.178]
  MoveL 308 to (229.26, 625.44, 0) mm, rotated rx 0 ry 90 rz -60.43 deg; joints [6.219, -39.823, 141.207, -54.748, -96.629, -9.277]
  MoveL 309 to (228.25, 627.85, 0) mm, rotated rx 0 ry 90 rz -60.43 deg; joints [6.085, -39.82, 141.293, -54.889, -96.659, -9.365]
  MoveL 310 to (227.46, 630.33, 0) mm, rotated rx 0 ry 90 rz -60.43 deg; joints [5.946, -39.817, 141.364, -55.035, -96.678, -9.441]
  MoveL 311 to (226.9, 632.88, 0) mm, rotated rx 0 ry 90 rz -60.43 deg; joints [5.801, -39.815, 141.42, -55.184, -96.687, -9.506]
  MoveL 312 to (226.56, 635.47, 0) mm, rotated rx 0 ry 90 rz -60.43 deg; joints [5.652, -39.814, 141.461, -55.336, -96.687, -9.558]
  MoveL 313 to (571.07, 677.93, 0) mm, rotated rx 0 ry 90 rz -60.43 deg; joints [2.344, -35.707, 116.085, -58.447, -84.93, 8.189]
  Set speed (60.0 mm/s)
  MoveL 314 to (569.05, 680.77, 0) mm, rotated rx 0 ry 90 rz -60.43 deg; joints [2.224, -35.757, 116.259, -58.557, -85.012, 8.093]
  MoveL 315 to (566.85, 683.46, 0) mm, rotated rx 0 ry 90 rz -60.43 deg; joints [2.111, -35.811, 116.446, -58.66, -85.098, 7.988]
  MoveL 316 to (564.48, 685.98, 0) mm, rotated rx 0 ry 90 rz -60.43 deg; joints [2.005, -35.868, 116.647, -58.755, -85.187, 7.875]
  MoveL 317 to (561.95, 688.35, 0) mm, rotated rx 0 ry 90 rz -60.43 deg; joints [1.906, -35.928, 116.859, -58.843, -85.279, 7.752]
  MoveL 318 to (559.27, 690.54, 0) mm, rotated rx 0 ry 90 rz -60.43 deg; joints [1.813, -35.991, 117.082, -58.923, -85.374, 7.623]
  MoveL 319 to (556.46, 692.56, 0) mm, rotated rx 0 ry 90 rz -60.43 deg; joints [1.729, -36.057, 117.315, -58.996, -85.471, 7.485]
  MoveL 320 to (553.52, 694.41, 0) mm, rotated rx 0 ry 90 rz -60.43 deg; joints [1.651, -36.124, 117.557, -59.061, -85.571, 7.341]
  MoveL 321 to (550.46, 696.07, 0) mm, rotated rx 0 ry 90 rz -60.43 deg; joints [1.582, -36.194, 117.807, -59.119, -85.673, 7.191]
  MoveL 322 to (547.32, 697.54, 0) mm, rotated rx 0 ry 90 rz -60.43 deg; joints [1.521, -36.265, 118.063, -59.168, -85.775, 7.036]
  MoveL 323 to (544.11, 698.82, 0) mm, rotated rx 0 ry 90 rz -60.43 deg; joints [1.468, -36.336, 118.324, -59.208, -85.879, 6.877]
  MoveL 324 to (540.83, 699.9, 0) mm, rotated rx 0 ry 90 rz -60.43 deg; joints [1.424, -36.409, 118.59, -59.241, -85.983, 6.713]
  MoveL 325 to (537.49, 700.79, 0) mm, rotated rx 0 ry 90 rz -60.43 deg; joints [1.388, -36.482, 118.859, -59.265, -86.087, 6.547]
  MoveL 326 to (534.1, 701.48, 0) mm, rotated rx 0 ry 90 rz -60.43 deg; joints [1.36, -36.555, 119.131, -59.28, -86.192, 6.377]
  MoveL 327 to (530.68, 701.98, 0) mm, rotated rx 0 ry 90 rz -60.43 deg; joints [1.342, -36.628, 119.405, -59.287, -86.296, 6.206]
  MoveL 328 to (527.24, 702.28, 0) mm, rotated rx 0 ry 90 rz -60.43 deg; joints [1.332, -36.701, 119.68, -59.286, -86.401, 6.032]
  MoveL 329 to (523.78, 702.38, 0) mm, rotated rx 0 ry 90 rz -60.43 deg; joints [1.331, -36.773, 119.955, -59.276, -86.504, 5.857]
  MoveL 330 to (361.71, 702.38, 0) mm, rotated rx 0 ry 90 rz -60.43 deg; joints [1.526, -39.291, 132.261, -58.937, -91.533, -2.543]
  MoveL 331 to (361.71, 740.48, 0) mm, rotated rx 0 ry 90 rz -60.43 deg; joints [-0.441, -39.295, 132.287, -60.903, -91.456, -2.614]
  MoveL 332 to (578.26, 740.48, 0) mm, rotated rx 0 ry 90 rz -60.43 deg; joints [-0.369, -35.561, 115.584, -61.168, -85.151, 8.73]
  MoveL 333 to (678.99, 588.08, 0) mm, rotated rx 0 ry 90 rz -60.43 deg; joints [5.756, -32.649, 106.405, -55.766, -80.691, 13.372]
  MoveL 334 to (630.46, 588.08, 0) mm, rotated rx 0 ry 90 rz -60.43 deg; joints [5.958, -34.033, 110.595, -55.22, -82.239, 11.004]
  MoveL 335 to (571.07, 677.93, 0) mm, rotated rx 0 ry 90 rz -60.43 deg; joints [2.344, -35.707, 116.085, -58.447, -84.93, 8.189]
  MoveL 336 to (437.55, 432.48, 0) mm, rotated rx 0 ry 90 rz -60.43 deg; joints [14.175, -37.724, 123.818, -46.32, -87.3, 2.824]
  Set speed (60.0 mm/s)
  MoveL 337 to (437.55, 470.58, 0) mm, rotated rx 0 ry 90 rz -60.43 deg; joints [12.431, -37.877, 124.493, -48.047, -87.736, 2.516]
  MoveL 338 to (247.79, 470.58, 0) mm, rotated rx 0 ry 90 rz -60.43 deg; joints [14.705, -39.806, 138.004, -46.017, -95.713, -5.889]
  MoveL 339 to (234.07, 472.17, 0) mm, rotated rx 0 ry 90 rz -60.43 deg; joints [14.815, -39.834, 138.954, -45.978, -96.366, -6.545]
  MoveL 340 to (227.45, 474.14, 0) mm, rotated rx 0 ry 90 rz -60.43 deg; joints [14.803, -39.841, 139.432, -46.029, -96.691, -6.887]
  MoveL 341 to (221.1, 476.88, 0) mm, rotated rx 0 ry 90 rz -60.43 deg; joints [14.744, -39.843, 139.903, -46.128, -97.01, -7.234]
  MoveL 342 to (215.11, 480.39, 0) mm, rotated rx 0 ry 90 rz -60.43 deg; joints [14.636, -39.84, 140.362, -46.278, -97.315, -7.584]
  MoveL 343 to (209.62, 484.61, 0) mm, rotated rx 0 ry 90 rz -60.43 deg; joints [14.48, -39.833, 140.799, -46.476, -97.6, -7.928]
  MoveL 344 to (204.72, 489.5, 0) mm, rotated rx 0 ry 90 rz -60.43 deg; joints [14.276, -39.823, 141.205, -46.721, -97.858, -8.261]
  MoveL 345 to (200.5, 495.02, 0) mm, rotated rx 0 ry 90 rz -60.43 deg; joints [14.023, -39.809, 141.575, -47.013, -98.083, -8.578]
  MoveL 346 to (73.96, 686.48, 0) mm, rotated rx 0 ry 90 rz -60.43 deg; joints [3.165, -37.762, 151.595, -59.542, -102.621, -20.383]
  MoveL 347 to (25.43, 686.48, 0) mm, rotated rx 0 ry 90 rz -60.43 deg; joints [3.363, -36.264, 154.524, -60.292, -104.917, -24.283]
  MoveL 348 to (193.3, 432.48, 0) mm, rotated rx 0 ry 90 rz -60.43 deg; joints [17.646, -39.831, 140.884, -43.317, -98.089, -7.558]
  MoveL 349 to (437.55, 432.48, 0) mm, rotated rx 0 ry 90 rz -60.43 deg; joints [14.175, -37.724, 123.818, -46.32, -87.3, 2.824]
  MoveL 350 to (528.52, 612.28, 0) mm, rotated rx 0 ry 90 rz -60.43 deg; joints [5.355, -36.562, 119.159, -55.298, -85.769, 6.081]
  Set speed (60.0 mm/s)
  MoveL 351 to (526.5, 615.11, 0) mm, rotated rx 0 ry 90 rz -60.43 deg; joints [5.237, -36.611, 119.34, -55.408, -85.857, 5.98]
  MoveL 352 to (524.3, 617.79, 0) mm, rotated rx 0 ry 90 rz -60.43 deg; joints [5.126, -36.662, 119.534, -55.51, -85.949, 5.87]
  MoveL 353 to (521.94, 620.32, 0) mm, rotated rx 0 ry 90 rz -60.43 deg; joints [5.023, -36.716, 119.74, -55.605, -86.045, 5.753]
  MoveL 354 to (519.41, 622.68, 0) mm, rotated rx 0 ry 90 rz -60.43 deg; joints [4.927, -36.773, 119.956, -55.691, -86.145, 5.627]
  MoveL 355 to (516.74, 624.87, 0) mm, rotated rx 0 ry 90 rz -60.43 deg; joints [4.838, -36.832, 120.182, -55.77, -86.248, 5.494]
  MoveL 356 to (513.93, 626.89, 0) mm, rotated rx 0 ry 90 rz -60.43 deg; joints [4.758, -36.893, 120.417, -55.841, -86.353, 5.355]
  MoveL 357 to (511, 628.74, 0) mm, rotated rx 0 ry 90 rz -60.43 deg; joints [4.686, -36.956, 120.66, -55.904, -86.461, 5.21]
  MoveL 358 to (507.91, 630.42, 0) mm, rotated rx 0 ry 90 rz -60.43 deg; joints [4.621, -37.02, 120.913, -55.959, -86.573, 5.057]
  MoveL 359 to (504.81, 631.87, 0) mm, rotated rx 0 ry 90 rz -60.43 deg; joints [4.566, -37.084, 121.166, -56.004, -86.683, 4.904]
  MoveL 360 to (501.59, 633.15, 0) mm, rotated rx 0 ry 90 rz -60.43 deg; joints [4.52, -37.15, 121.426, -56.042, -86.796, 4.745]
  MoveL 361 to (498.3, 634.24, 0) mm, rotated rx 0 ry 90 rz -60.43 deg; joints [4.482, -37.215, 121.69, -56.07, -86.909, 4.582]
  MoveL 362 to (494.96, 635.13, 0) mm, rotated rx 0 ry 90 rz -60.43 deg; joints [4.453, -37.281, 121.957, -56.09, -87.024, 4.417]
  MoveL 363 to (491.57, 635.82, 0) mm, rotated rx 0 ry 90 rz -60.43 deg; joints [4.433, -37.347, 122.225, -56.101, -87.138, 4.249]
  MoveL 364 to (488.14, 636.32, 0) mm, rotated rx 0 ry 90 rz -60.43 deg; joints [4.423, -37.412, 122.495, -56.104, -87.253, 4.08]
  MoveL 365 to (484.69, 636.62, 0) mm, rotated rx 0 ry 90 rz -60.43 deg; joints [4.421, -37.477, 122.765, -56.097, -87.367, 3.91]
  MoveL 366 to (481.23, 636.72, 0) mm, rotated rx 0 ry 90 rz -60.43 deg; joints [4.429, -37.541, 123.034, -56.082, -87.481, 3.739]
  MoveL 367 to (269.9, 636.72, 0) mm, rotated rx 0 ry 90 rz -60.43 deg; joints [5.343, -39.823, 138.503, -55.394, -94.955, -7.136]
  MoveL 368 to (269.9, 674.82, 0) mm, rotated rx 0 ry 90 rz -60.43 deg; joints [3.211, -39.828, 138.701, -57.53, -94.79, -7.477]
  MoveL 369 to (535.71, 674.82, 0) mm, rotated rx 0 ry 90 rz -60.43 deg; joints [2.547, -36.501, 118.93, -58.107, -85.983, 6.423]
  MoveL 370 to (636.44, 522.42, 0) mm, rotated rx 0 ry 90 rz -60.43 deg; joints [8.605, -33.638, 109.372, -52.692, -81.239, 11.303]
  MoveL 371 to (587.91, 522.42, 0) mm, rotated rx 0 ry 90 rz -60.43 deg; joints [8.913, -34.921, 113.438, -52.079, -82.883, 9.036]
  MoveL 372 to (528.52, 612.28, 0) mm, rotated rx 0 ry 90 rz -60.43 deg; joints [5.355, -36.562, 119.159, -55.298, -85.769, 6.081]
  MoveL 373 to (1077.92, 419.21, 0) mm, rotated rx 0 ry 90 rz -60.43 deg; joints [9.718, -13.48, 59.238, -59.623, -63.781, 37.007]
  Set speed (60.0 mm/s)
  MoveL 374 to (1116.02, 419.21, 0) mm, rotated rx 0 ry 90 rz -60.43 deg; joints [9.523, -10.561, 52.803, -61.355, -62.171, 40.518]
  MoveL 375 to (1116.02, 663.46, 0) mm, rotated rx 0 ry 90 rz -60.43 deg; joints [2.104, -12.536, 57.144, -66.573, -68.048, 40.786]
  MoveL 376 to (862.02, 663.46, 0) mm, rotated rx 0 ry 90 rz -60.43 deg; joints [2.435, -26.383, 89.503, -60.86, -76.135, 23.259]
  MoveL 377 to (862.02, 612.51, 0) mm, rotated rx 0 ry 90 rz -60.43 deg; joints [4.242, -26.26, 89.195, -59.187, -75.332, 23.003]
  MoveL 378 to (1027.12, 612.51, 0) mm, rotated rx 0 ry 90 rz -60.43 deg; joints [3.849, -18.218, 69.94, -62.615, -70.05, 33.371]
  MoveL 379 to (1032.37, 612.21, 0) mm, rotated rx 0 ry 90 rz -60.43 deg; joints [3.847, -17.91, 69.233, -62.746, -69.868, 33.749]
  MoveL 380 to (1037.49, 611.35, 0) mm, rotated rx 0 ry 90 rz -60.43 deg; joints [3.864, -17.604, 68.53, -62.861, -69.678, 34.119]
  MoveL 381 to (1042.45, 609.93, 0) mm, rotated rx 0 ry 90 rz -60.43 deg; joints [3.898, -17.3, 67.837, -62.96, -69.481, 34.479]
  MoveL 382 to (1047.22, 608, 0) mm, rotated rx 0 ry 90 rz -60.43 deg; joints [3.949, -17.002, 67.158, -63.043, -69.279, 34.826]
  MoveL 383 to (1051.75, 605.57, 0) mm, rotated rx 0 ry 90 rz -60.43 deg; joints [4.016, -16.712, 66.499, -63.109, -69.073, 35.158]
  MoveL 384 to (1056.03, 602.67, 0) mm, rotated rx 0 ry 90 rz -60.43 deg; joints [4.098, -16.432, 65.864, -63.159, -68.865, 35.471]
  MoveL 385 to (1060.02, 599.34, 0) mm, rotated rx 0 ry 90 rz -60.43 deg; joints [4.194, -16.165, 65.258, -63.193, -68.657, 35.765]
  MoveL 386 to (1063.69, 595.59, 0) mm, rotated rx 0 ry 90 rz -60.43 deg; joints [4.304, -15.913, 64.689, -63.209, -68.449, 36.034]
  MoveL 387 to (1066.98, 591.48, 0) mm, rotated rx 0 ry 90 rz -60.43 deg; joints [4.425, -15.68, 64.163, -63.207, -68.246, 36.277]
  MoveL 388 to (1069.85, 587.11, 0) mm, rotated rx 0 ry 90 rz -60.43 deg; joints [4.555, -15.471, 63.691, -63.189, -68.05, 36.487]
  MoveL 389 to (1072.29, 582.5, 0) mm, rotated rx 0 ry 90 rz -60.43 deg; joints [4.693, -15.285, 63.274, -63.153, -67.863, 36.666]
  MoveL 390 to (1074.3, 577.69, 0) mm, rotated rx 0 ry 90 rz -60.43 deg; joints [4.838, -15.125, 62.914, -63.1, -67.686, 36.81]
  MoveL 391 to (1075.88, 572.71, 0) mm, rotated rx 0 ry 90 rz -60.43 deg; joints [4.989, -14.992, 62.614, -63.03, -67.52, 36.921]
  MoveL 392 to (1077.01, 567.62, 0) mm, rotated rx 0 ry 90 rz -60.43 deg; joints [5.145, -14.885, 62.376, -62.945, -67.367, 36.997]
  MoveL 393 to (1077.69, 562.43, 0) mm, rotated rx 0 ry 90 rz -60.43 deg; joints [5.304, -14.807, 62.201, -62.843, -67.227, 37.037]
  MoveL 394 to (1077.92, 557.19, 0) mm, rotated rx 0 ry 90 rz -60.43 deg; joints [5.466, -14.759, 62.091, -62.725, -67.101, 37.041]
  MoveL 395 to (1077.92, 419.21, 0) mm, rotated rx 0 ry 90 rz -60.43 deg; joints [9.718, -13.48, 59.238, -59.623, -63.781, 37.007]
  MoveL 396 to (169.13, 240.44, 0) mm, rotated rx 0 ry 90 rz -60.43 deg; joints [28.185, -39.77, 137.233, -32.463, -96.308, -3.998]
  Set speed (60.0 mm/s)
  MoveL 397 to (165.77, 242.52, 0) mm, rotated rx 0 ry 90 rz -60.43 deg; joints [28.172, -39.784, 137.51, -32.493, -96.528, -4.141]
  MoveL 398 to (162.31, 244.16, 0) mm, rotated rx 0 ry 90 rz -60.43 deg; joints [28.182, -39.796, 137.778, -32.499, -96.744, -4.278]
  MoveL 399 to (158.78, 245.34, 0) mm, rotated rx 0 ry 90 rz -60.43 deg; joints [28.217, -39.807, 138.034, -32.479, -96.954, -4.407]
  MoveL 400 to (155.16, 246.02, 0) mm, rotated rx 0 ry 90 rz -60.43 deg; joints [28.279, -39.816, 138.279, -32.433, -97.158, -4.527]
  MoveL 401 to (151.46, 246.17, 0) mm, rotated rx 0 ry 90 rz -60.43 deg; joints [28.37, -39.823, 138.51, -32.357, -97.355, -4.637]
  MoveL 402 to (147.69, 245.75, 0) mm, rotated rx 0 ry 90 rz -60.43 deg; joints [28.492, -39.829, 138.726, -32.249, -97.542, -4.734]
  MoveL 403 to (143.86, 244.72, 0) mm, rotated rx 0 ry 90 rz -60.43 deg; joints [28.645, -39.833, 138.926, -32.108, -97.72, -4.818]
  MoveL 404 to (139.97, 243.06, 0) mm, rotated rx 0 ry 90 rz -60.43 deg; joints [28.833, -39.837, 139.107, -31.932, -97.887, -4.888]
  MoveL 405 to (136.02, 240.72, 0) mm, rotated rx 0 ry 90 rz -60.43 deg; joints [29.057, -39.839, 139.268, -31.719, -98.04, -4.941]
  MoveL 406 to (132.02, 237.68, 0) mm, rotated rx 0 ry 90 rz -60.43 deg; joints [29.318, -39.841, 139.406, -31.466, -98.179, -4.976]
  MoveL 407 to (127.98, 233.89, 0) mm, rotated rx 0 ry 90 rz -60.43 deg; joints [29.619, -39.842, 139.521, -31.172, -98.303, -4.992]
  MoveL 408 to (122.21, 227.21, 0) mm, rotated rx 0 ry 90 rz -60.43 deg; joints [30.112, -39.842, 139.636, -30.685, -98.444, -4.98]
  MoveL 409 to (117.01, 219.8, 0) mm, rotated rx 0 ry 90 rz -60.43 deg; joints [30.626, -39.843, 139.687, -30.17, -98.532, -4.929]
  MoveL 410 to (112.37, 212, 0) mm, rotated rx 0 ry 90 rz -60.43 deg; joints [31.143, -39.843, 139.685, -29.649, -98.575, -4.851]
  MoveL 411 to (108.32, 204.19, 0) mm, rotated rx 0 ry 90 rz -60.43 deg; joints [31.643, -39.842, 139.643, -29.142, -98.58, -4.755]
  MoveL 412 to (104.31, 195.46, 0) mm, rotated rx 0 ry 90 rz -60.43 deg; joints [32.186, -39.842, 139.56, -28.589, -98.552, -4.633]
  MoveL 413 to (100.58, 186.36, 0) mm, rotated rx 0 ry 90 rz -60.43 deg; joints [32.736, -39.841, 139.44, -28.026, -98.491, -4.494]
  MoveL 414 to (93.92, 167.42, 0) mm, rotated rx 0 ry 90 rz -60.43 deg; joints [33.84, -39.837, 139.106, -26.891, -98.282, -4.178]
  MoveL 415 to (88.29, 148.15, 0) mm, rotated rx 0 ry 90 rz -60.43 deg; joints [34.915, -39.827, 138.674, -25.781, -97.978, -3.835]
  MoveL 416 to (83.64, 129.34, 0) mm, rotated rx 0 ry 90 rz -60.43 deg; joints [35.925, -39.812, 138.18, -24.736, -97.609, -3.491]
  MoveL 417 to (82.2, 122.92, 0) mm, rotated rx 0 ry 90 rz -60.43 deg; joints [36.261, -39.805, 137.997, -24.388, -97.469, -3.373]
  MoveL 418 to (77.52, 99.15, 0) mm, rotated rx 0 ry 90 rz -60.43 deg; joints [37.469, -39.771, 137.261, -23.136, -96.893, -2.936]
  MoveL 419 to (73.6, 74.87, 0) mm, rotated rx 0 ry 90 rz -60.43 deg; joints [38.648, -39.72, 136.424, -21.916, -96.224, -2.497]
  MoveL 420 to (70.4, 50.34, 0) mm, rotated rx 0 ry 90 rz -60.43 deg; joints [39.786, -39.649, 135.501, -20.741, -95.475, -2.069]
  MoveL 421 to (67.87, 25.85, 0) mm, rotated rx 0 ry 90 rz -60.43 deg; joints [40.872, -39.557, 134.508, -19.624, -94.665, -1.661]
  MoveL 422 to (63.5, 25.44, 0) mm, rotated rx 0 ry 90 rz -60.43 deg; joints [41.041, -39.578, 134.725, -19.46, -94.854, -1.713]
  MoveL 423 to (25.4, 25.44, 0) mm, rotated rx 0 ry 90 rz -60.43 deg; joints [42.409, -39.741, 136.743, -18.146, -96.657, -2.176]
  MoveL 424 to (25.4, 591.47, 0) mm, rotated rx 0 ry 90 rz -60.43 deg; joints [10.293, -36.659, 153.852, -53.396, -107.033, -21.522]
  MoveL 425 to (434.22, 25.44, 0) mm, rotated rx 0 ry 90 rz -60.43 deg; joints [30.861, -34.268, 111.336, -30.203, -78.775, 6.465]
  MoveL 426 to (404.04, 32.53, 0) mm, rotated rx 0 ry 90 rz -60.43 deg; joints [31.26, -35.035, 113.814, -29.641, -80.217, 5.523]
  MoveL 427 to (373.28, 38.93, 0) mm, rotated rx 0 ry 90 rz -60.43 deg; joints [31.716, -35.754, 116.25, -29.047, -81.673, 4.598]
  MoveL 428 to (342.35, 44.38, 0) mm, rotated rx 0 ry 90 rz -60.43 deg; joints [32.233, -36.413, 118.607, -28.418, -83.124, 3.706]
  MoveL 429 to (311.63, 48.63, 0) mm, rotated rx 0 ry 90 rz -60.43 deg; joints [32.815, -37.004, 120.848, -27.75, -84.548, 2.862]
  MoveL 430 to (184.4, 224.78, 0) mm, rotated rx 0 ry 90 rz -60.43 deg; joints [28.541, -39.671, 135.76, -32.033, -95.168, -3.226]
  MoveL 431 to (178.62, 231.96, 0) mm, rotated rx 0 ry 90 rz -60.43 deg; joints [28.348, -39.716, 136.362, -32.254, -95.628, -3.541]
  MoveL 432 to (172.4, 237.96, 0) mm, rotated rx 0 ry 90 rz -60.43 deg; joints [28.22, -39.754, 136.949, -32.413, -96.084, -3.85]
  MoveL 433 to (169.13, 240.44, 0) mm, rotated rx 0 ry 90 rz -60.43 deg; joints [28.185, -39.77, 137.233, -32.463, -96.308, -3.998]
  MoveL 434 to (740.63, 520.58, 0) mm, rotated rx 0 ry 90 rz -60.43 deg; joints [8.08, -30.429, 100.111, -54.113, -77.754, 16.338]
  Set speed (60.0 mm/s)
  MoveL 435 to (743.25, 520.7, 0) mm, rotated rx 0 ry 90 rz -60.43 deg; joints [8.062, -30.341, 99.871, -54.158, -77.67, 16.469]
  MoveL 436 to (791.49, 520.7, 0) mm, rotated rx 0 ry 90 rz -60.43 deg; joints [7.812, -28.636, 95.3, -54.946, -76.084, 18.921]
  MoveL 437 to (798.37, 519.9, 0) mm, rotated rx 0 ry 90 rz -60.43 deg; joints [7.807, -28.377, 94.621, -55.037, -75.845, 19.277]
  MoveL 438 to (801.68, 518.91, 0) mm, rotated rx 0 ry 90 rz -60.43 deg; joints [7.827, -28.248, 94.284, -55.061, -75.719, 19.448]
  MoveL 439 to (804.85, 517.54, 0) mm, rotated rx 0 ry 90 rz -60.43 deg; joints [7.86, -28.122, 93.956, -55.071, -75.592, 19.611]
  MoveL 440 to (807.82, 515.81, 0) mm, rotated rx 0 ry 90 rz -60.43 deg; joints [7.908, -28, 93.64, -55.066, -75.465, 19.764]
  MoveL 441 to (810.55, 513.71, 0) mm, rotated rx 0 ry 90 rz -60.43 deg; joints [7.97, -27.885, 93.341, -55.045, -75.338, 19.904]
  MoveL 442 to (813.01, 511.27, 0) mm, rotated rx 0 ry 90 rz -60.43 deg; joints [8.046, -27.778, 93.064, -55.008, -75.215, 20.029]
  MoveL 443 to (815.14, 508.48, 0) mm, rotated rx 0 ry 90 rz -60.43 deg; joints [8.135, -27.681, 92.814, -54.954, -75.096, 20.137]
  MoveL 444 to (916.18, 355.6, 0) mm, rotated rx 0 ry 90 rz -60.43 deg; joints [12.742, -22.118, 79.061, -52.656, -68.457, 25.7]
  MoveL 445 to (964.71, 355.6, 0) mm, rotated rx 0 ry 90 rz -60.43 deg; joints [12.392, -19.66, 73.273, -54.098, -66.63, 28.72]
  MoveL 446 to (830.41, 558.8, 0) mm, rotated rx 0 ry 90 rz -60.43 deg; joints [6.259, -27.334, 91.922, -56.888, -75.451, 21.066]
  MoveL 447 to (664.63, 558.8, 0) mm, rotated rx 0 ry 90 rz -60.43 deg; joints [6.987, -32.976, 107.374, -54.465, -80.781, 12.643]
  MoveL 448 to (664.63, 254, 0) mm, rotated rx 0 ry 90 rz -60.43 deg; joints [18.691, -30.842, 101.251, -43.439, -75.51, 13.33]
  MoveL 449 to (715.59, 254, 0) mm, rotated rx 0 ry 90 rz -60.43 deg; joints [18.084, -29.16, 96.687, -44.604, -73.589, 15.57]
  MoveL 450 to (715.59, 495.3, 0) mm, rotated rx 0 ry 90 rz -60.43 deg; joints [9.184, -31.13, 102.052, -52.814, -78.193, 15.094]
  MoveL 451 to (715.73, 497.93, 0) mm, rotated rx 0 ry 90 rz -60.43 deg; joints [9.083, -31.139, 102.077, -52.911, -78.229, 15.101]
  MoveL 452 to (716.17, 500.49, 0) mm, rotated rx 0 ry 90 rz -60.43 deg; joints [8.982, -31.138, 102.074, -53.011, -78.255, 15.123]
  MoveL 453 to (716.88, 502.97, 0) mm, rotated rx 0 ry 90 rz -60.43 deg; joints [8.883, -31.127, 102.045, -53.111, -78.269, 15.157]
  MoveL 454 to (717.84, 505.35, 0) mm, rotated rx 0 ry 90 rz -60.43 deg; joints [8.787, -31.108, 101.991, -53.212, -78.274, 15.205]
  MoveL 455 to (719.06, 507.62, 0) mm, rotated rx 0 ry 90 rz -60.43 deg; joints [8.693, -31.08, 101.913, -53.313, -78.268, 15.265]
  MoveL 456 to (720.51, 509.76, 0) mm, rotated rx 0 ry 90 rz -60.43 deg; joints [8.603, -31.043, 101.811, -53.413, -78.253, 15.337]
  MoveL 457 to (722.17, 511.75, 0) mm, rotated rx 0 ry 90 rz -60.43 deg; joints [8.517, -30.999, 101.686, -53.51, -78.228, 15.42]
  MoveL 458 to (724.05, 513.58, 0) mm, rotated rx 0 ry 90 rz -60.43 deg; joints [8.437, -30.946, 101.54, -53.605, -78.194, 15.513]
  MoveL 459 to (726.1, 515.23, 0) mm, rotated rx 0 ry 90 rz -60.43 deg; joints [8.363, -30.887, 101.375, -53.696, -78.151, 15.615]
  MoveL 460 to (728.29, 516.66, 0) mm, rotated rx 0 ry 90 rz -60.43 deg; joints [8.296, -30.822, 101.195, -53.781, -78.101, 15.723]
  MoveL 461 to (730.59, 517.89, 0) mm, rotated rx 0 ry 90 rz -60.43 deg; joints [8.237, -30.751, 101, -53.861, -78.044, 15.838]
  MoveL 462 to (733, 518.89, 0) mm, rotated rx 0 ry 90 rz -60.43 deg; joints [8.185, -30.676, 100.792, -53.934, -77.98, 15.958]
  MoveL 463 to (735.49, 519.68, 0) mm, rotated rx 0 ry 90 rz -60.43 deg; joints [8.142, -30.597, 100.574, -54.001, -77.91, 16.082]
  MoveL 464 to (738.03, 520.24, 0) mm, rotated rx 0 ry 90 rz -60.43 deg; joints [8.107, -30.514, 100.346, -54.06, -77.834, 16.209]
  MoveL 465 to (740.63, 520.58, 0) mm, rotated rx 0 ry 90 rz -60.43 deg; joints [8.08, -30.429, 100.111, -54.113, -77.754, 16.338]
  MoveL 466 to (531.29, 471.54, 0) mm, rotated rx 0 ry 90 rz -60.43 deg; joints [11.505, -36.046, 117.277, -49.257, -84.251, 6.633]
  Set speed (60.0 mm/s)
  MoveL 467 to (529.27, 474.38, 0) mm, rotated rx 0 ry 90 rz -60.43 deg; joints [11.4, -36.104, 117.483, -49.35, -84.359, 6.53]
  MoveL 468 to (527.07, 477.06, 0) mm, rotated rx 0 ry 90 rz -60.43 deg; joints [11.303, -36.164, 117.7, -49.435, -84.472, 6.42]
  MoveL 469 to (524.7, 479.59, 0) mm, rotated rx 0 ry 90 rz -60.43 deg; joints [11.214, -36.227, 117.927, -49.512, -84.589, 6.303]
  MoveL 470 to (522.17, 481.95, 0) mm, rotated rx 0 ry 90 rz -60.43 deg; joints [11.134, -36.292, 118.164, -49.581, -84.709, 6.18]
  MoveL 471 to (519.49, 484.15, 0) mm, rotated rx 0 ry 90 rz -60.43 deg; joints [11.061, -36.36, 118.409, -49.641, -84.832, 6.05]
  MoveL 472 to (516.68, 486.17, 0) mm, rotated rx 0 ry 90 rz -60.43 deg; joints [10.997, -36.428, 118.661, -49.692, -84.958, 5.915]
  MoveL 473 to (513.74, 488.02, 0) mm, rotated rx 0 ry 90 rz -60.43 deg; joints [10.941, -36.498, 118.921, -49.736, -85.086, 5.775]
  MoveL 474 to (510.68, 489.68, 0) mm, rotated rx 0 ry 90 rz -60.43 deg; joints [10.894, -36.569, 119.186, -49.77, -85.216, 5.631]
  MoveL 475 to (507.54, 491.15, 0) mm, rotated rx 0 ry 90 rz -60.43 deg; joints [10.856, -36.641, 119.454, -49.796, -85.346, 5.483]
  MoveL 476 to (504.33, 492.42, 0) mm, rotated rx 0 ry 90 rz -60.43 deg; joints [10.827, -36.712, 119.724, -49.813, -85.477, 5.333]
  MoveL 477 to (501.05, 493.51, 0) mm, rotated rx 0 ry 90 rz -60.43 deg; joints [10.806, -36.784, 119.996, -49.821, -85.609, 5.181]
  MoveL 478 to (497.71, 494.4, 0) mm, rotated rx 0 ry 90 rz -60.43 deg; joints [10.795, -36.855, 120.27, -49.82, -85.74, 5.027]
  MoveL 479 to (494.32, 495.09, 0) mm, rotated rx 0 ry 90 rz -60.43 deg; joints [10.793, -36.926, 120.543, -49.811, -85.871, 4.872]
  MoveL 480 to (490.9, 495.58, 0) mm, rotated rx 0 ry 90 rz -60.43 deg; joints [10.8, -36.995, 120.816, -49.793, -86.002, 4.716]
  MoveL 481 to (487.46, 495.88, 0) mm, rotated rx 0 ry 90 rz -60.43 deg; joints [10.816, -37.064, 121.087, -49.766, -86.131, 4.56]
  MoveL 482 to (484, 495.98, 0) mm, rotated rx 0 ry 90 rz -60.43 deg; joints [10.841, -37.132, 121.356, -49.731, -86.259, 4.404]
  MoveL 483 to (289.09, 495.98, 0) mm, rotated rx 0 ry 90 rz -60.43 deg; joints [12.817, -39.658, 135.604, -47.766, -94.005, -4.399]
  MoveL 484 to (289.09, 534.08, 0) mm, rotated rx 0 ry 90 rz -60.43 deg; joints [10.8, -39.701, 136.157, -49.808, -94.177, -4.927]
  MoveL 485 to (538.48, 534.08, 0) mm, rotated rx 0 ry 90 rz -60.43 deg; joints [8.743, -36.135, 117.593, -51.996, -84.717, 6.721]
  MoveL 486 to (639.21, 381.68, 0) mm, rotated rx 0 ry 90 rz -60.43 deg; joints [14.17, -32.753, 106.712, -47.394, -78.986, 11.735]
  MoveL 487 to (590.68, 381.68, 0) mm, rotated rx 0 ry 90 rz -60.43 deg; joints [14.662, -34.093, 110.783, -46.546, -80.758, 9.621]
  MoveL 488 to (531.29, 471.54, 0) mm, rotated rx 0 ry 90 rz -60.43 deg; joints [11.505, -36.046, 117.277, -49.257, -84.251, 6.633]
  MoveL 489 to (715.95, 227.1, 0) mm, rotated rx 0 ry 90 rz -60.43 deg; joints [19.026, -28.835, 95.825, -43.769, -72.95, 15.688]
  Set speed (60.0 mm/s)
  MoveL 490 to (713.33, 226.99, 0) mm, rotated rx 0 ry 90 rz -60.43 deg; joints [19.061, -28.924, 96.062, -43.702, -73.047, 15.571]
  MoveL 491 to (665.08, 226.99, 0) mm, rotated rx 0 ry 90 rz -60.43 deg; joints [19.663, -30.53, 100.389, -42.561, -74.883, 13.468]
  MoveL 492 to (658.2, 227.79, 0) mm, rotated rx 0 ry 90 rz -60.43 deg; joints [19.723, -30.757, 101.015, -42.428, -75.163, 13.173]
  MoveL 493 to (654.89, 228.77, 0) mm, rotated rx 0 ry 90 rz -60.43 deg; joints [19.73, -30.872, 101.334, -42.385, -75.312, 13.029]
  MoveL 494 to (651.73, 230.14, 0) mm, rotated rx 0 ry 90 rz -60.43 deg; joints [19.722, -30.986, 101.651, -42.358, -75.464, 12.89]
  MoveL 495 to (648.76, 231.88, 0) mm, rotated rx 0 ry 90 rz -60.43 deg; joints [19.697, -31.098, 101.962, -42.348, -75.617, 12.757]
  MoveL 496 to (646.02, 233.97, 0) mm, rotated rx 0 ry 90 rz -60.43 deg; joints [19.656, -31.205, 102.263, -42.355, -75.769, 12.633]
  MoveL 497 to (643.57, 236.42, 0) mm, rotated rx 0 ry 90 rz -60.43 deg; joints [19.599, -31.307, 102.55, -42.382, -75.918, 12.519]
  MoveL 498 to (641.44, 239.21, 0) mm, rotated rx 0 ry 90 rz -60.43 deg; joints [19.525, -31.403, 102.818, -42.427, -76.061, 12.416]
  MoveL 499 to (540.39, 392.09, 0) mm, rotated rx 0 ry 90 rz -60.43 deg; joints [14.776, -35.412, 115.076, -46.121, -82.795, 7.431]
  MoveL 500 to (491.86, 392.09, 0) mm, rotated rx 0 ry 90 rz -60.43 deg; joints [15.327, -36.488, 118.881, -45.354, -84.639, 5.404]
  MoveL 501 to (626.16, 188.89, 0) mm, rotated rx 0 ry 90 rz -60.43 deg; joints [21.562, -31.294, 102.512, -40.406, -75.482, 12.046]
  MoveL 502 to (791.94, 188.89, 0) mm, rotated rx 0 ry 90 rz -60.43 deg; joints [19.424, -25.484, 87.252, -44.62, -69.085, 19.406]
  MoveL 503 to (791.94, 493.69, 0) mm, rotated rx 0 ry 90 rz -60.43 deg; joints [8.794, -28.473, 94.875, -54.042, -75.613, 18.908]
  MoveL 504 to (740.99, 493.69, 0) mm, rotated rx 0 ry 90 rz -60.43 deg; joints [9.09, -30.279, 99.702, -53.166, -77.316, 16.338]
  MoveL 505 to (740.99, 252.39, 0) mm, rotated rx 0 ry 90 rz -60.43 deg; joints [17.851, -28.246, 94.28, -45.157, -72.596, 16.739]
  MoveL 506 to (740.84, 249.76, 0) mm, rotated rx 0 ry 90 rz -60.43 deg; joints [17.944, -28.221, 94.214, -45.073, -72.54, 16.741]
  MoveL 507 to (740.41, 247.2, 0) mm, rotated rx 0 ry 90 rz -60.43 deg; joints [18.038, -28.206, 94.177, -44.984, -72.497, 16.73]
  MoveL 508 to (739.7, 244.72, 0) mm, rotated rx 0 ry 90 rz -60.43 deg; joints [18.133, -28.203, 94.167, -44.89, -72.466, 16.706]
  MoveL 509 to (738.73, 242.34, 0) mm, rotated rx 0 ry 90 rz -60.43 deg; joints [18.227, -28.209, 94.184, -44.793, -72.446, 16.669]
  MoveL 510 to (737.52, 240.07, 0) mm, rotated rx 0 ry 90 rz -60.43 deg; joints [18.319, -28.226, 94.228, -44.694, -72.439, 16.621]
  MoveL 511 to (736.07, 237.93, 0) mm, rotated rx 0 ry 90 rz -60.43 deg; joints [18.41, -28.253, 94.297, -44.593, -72.443, 16.562]
  MoveL 512 to (734.4, 235.93, 0) mm, rotated rx 0 ry 90 rz -60.43 deg; joints [18.499, -28.289, 94.391, -44.491, -72.459, 16.493]
  MoveL 513 to (732.53, 234.1, 0) mm, rotated rx 0 ry 90 rz -60.43 deg; joints [18.585, -28.334, 94.509, -44.389, -72.487, 16.413]
  MoveL 514 to (730.47, 232.45, 0) mm, rotated rx 0 ry 90 rz -60.43 deg; joints [18.666, -28.387, 94.649, -44.288, -72.526, 16.326]
  MoveL 515 to (728.29, 231.02, 0) mm, rotated rx 0 ry 90 rz -60.43 deg; joints [18.742, -28.448, 94.807, -44.191, -72.575, 16.231]
  MoveL 516 to (725.98, 229.8, 0) mm, rotated rx 0 ry 90 rz -60.43 deg; joints [18.811, -28.515, 94.983, -44.097, -72.633, 16.131]
  MoveL 517 to (723.58, 228.79, 0) mm, rotated rx 0 ry 90 rz -60.43 deg; joints [18.875, -28.588, 95.174, -44.007, -72.701, 16.026]
  MoveL 518 to (721.09, 228.01, 0) mm, rotated rx 0 ry 90 rz -60.43 deg; joints [18.932, -28.666, 95.379, -43.922, -72.777, 15.916]
  MoveL 519 to (718.54, 227.44, 0) mm, rotated rx 0 ry 90 rz -60.43 deg; joints [18.982, -28.748, 95.597, -43.842, -72.86, 15.803]
  MoveL 520 to (715.95, 227.1, 0) mm, rotated rx 0 ry 90 rz -60.43 deg; joints [19.026, -28.835, 95.825, -43.769, -72.95, 15.688]
  MoveL 521 to (444.31, 344.54, 0) mm, rotated rx 0 ry 90 rz -60.43 deg; joints [17.999, -37.146, 121.413, -42.573, -85.771, 3.875]
  Set speed (60.0 mm/s)
  MoveL 522 to (442.29, 347.38, 0) mm, rotated rx 0 ry 90 rz -60.43 deg; joints [17.904, -37.201, 121.632, -42.66, -85.899, 3.77]
  MoveL 523 to (440.09, 350.06, 0) mm, rotated rx 0 ry 90 rz -60.43 deg; joints [17.817, -37.258, 121.861, -42.738, -86.031, 3.66]
  MoveL 524 to (435.19, 354.95, 0) mm, rotated rx 0 ry 90 rz -60.43 deg; joints [17.672, -37.375, 122.342, -42.867, -86.307, 3.422]
  MoveL 525 to (429.7, 359.17, 0) mm, rotated rx 0 ry 90 rz -60.43 deg; joints [17.563, -37.497, 122.849, -42.96, -86.595, 3.166]
  MoveL 526 to (423.7, 362.68, 0) mm, rotated rx 0 ry 90 rz -60.43 deg; joints [17.491, -37.621, 123.375, -43.016, -86.893, 2.895]
  MoveL 527 to (417.35, 365.42, 0) mm, rotated rx 0 ry 90 rz -60.43 deg; joints [17.458, -37.744, 123.907, -43.035, -87.193, 2.618]
  MoveL 528 to (410.73, 367.39, 0) mm, rotated rx 0 ry 90 rz -60.43 deg; joints [17.463, -37.865, 124.439, -43.017, -87.494, 2.336]
  MoveL 529 to (403.93, 368.58, 0) mm, rotated rx 0 ry 90 rz -60.43 deg; joints [17.506, -37.981, 124.965, -42.962, -87.791, 2.055]
  MoveL 530 to (397.02, 368.98, 0) mm, rotated rx 0 ry 90 rz -60.43 deg; joints [17.587, -38.092, 125.477, -42.871, -88.083, 1.779]
  MoveL 531 to (223.67, 368.98, 0) mm, rotated rx 0 ry 90 rz -60.43 deg; joints [20.481, -39.782, 137.463, -40.202, -95.882, -4.95]
  MoveL 532 to (223.67, 407.08, 0) mm, rotated rx 0 ry 90 rz -60.43 deg; joints [18.485, -39.818, 138.351, -42.261, -96.336, -5.727]
  MoveL 533 to (451.51, 407.08, 0) mm, rotated rx 0 ry 90 rz -60.43 deg; joints [15.153, -37.358, 122.27, -45.389, -86.422, 3.619]
  MoveL 534 to (619.38, 153.08, 0) mm, rotated rx 0 ry 90 rz -60.43 deg; joints [22.943, -31.055, 101.844, -39.081, -74.864, 11.972]
  MoveL 535 to (570.85, 153.08, 0) mm, rotated rx 0 ry 90 rz -60.43 deg; joints [23.696, -32.466, 105.868, -37.908, -76.766, 10.108]
  MoveL 536 to (444.31, 344.54, 0) mm, rotated rx 0 ry 90 rz -60.43 deg; joints [17.999, -37.146, 121.413, -42.573, -85.771, 3.875]
  MoveL 537 to (791.94, 89.58, 0) mm, rotated rx 0 ry 90 rz -60.43 deg; joints [22.642, -23.906, 83.37, -41.992, -66.325, 19.873]
  Set speed (60.0 mm/s)
  MoveL 538 to (791.94, 127.68, 0) mm, rotated rx 0 ry 90 rz -60.43 deg; joints [21.424, -24.552, 84.947, -42.97, -67.425, 19.677]
  MoveL 539 to (569.33, 127.68, 0) mm, rotated rx 0 ry 90 rz -60.43 deg; joints [24.64, -32.19, 105.065, -37.03, -76.181, 10.214]
  MoveL 540 to (555.62, 129.27, 0) mm, rotated rx 0 ry 90 rz -60.43 deg; joints [24.81, -32.59, 106.231, -36.746, -76.764, 9.701]
  MoveL 541 to (549, 131.24, 0) mm, rotated rx 0 ry 90 rz -60.43 deg; joints [24.85, -32.795, 106.834, -36.651, -77.077, 9.447]
  MoveL 542 to (542.65, 133.98, 0) mm, rotated rx 0 ry 90 rz -60.43 deg; joints [24.857, -32.999, 107.442, -36.589, -77.399, 9.199]
  MoveL 543 to (536.65, 137.49, 0) mm, rotated rx 0 ry 90 rz -60.43 deg; joints [24.83, -33.201, 108.045, -36.564, -77.727, 8.96]
  MoveL 544 to (531.16, 141.71, 0) mm, rotated rx 0 ry 90 rz -60.43 deg; joints [24.768, -33.395, 108.632, -36.576, -78.052, 8.734]
  MoveL 545 to (526.26, 146.6, 0) mm, rotated rx 0 ry 90 rz -60.43 deg; joints [24.671, -33.579, 109.194, -36.628, -78.369, 8.524]
  MoveL 546 to (522.04, 152.12, 0) mm, rotated rx 0 ry 90 rz -60.43 deg; joints [24.537, -33.752, 109.722, -36.719, -78.674, 8.334]
  MoveL 547 to (395.5, 343.58, 0) mm, rotated rx 0 ry 90 rz -60.43 deg; joints [18.757, -37.985, 124.982, -41.71, -87.757, 1.998]
  MoveL 548 to (346.97, 343.58, 0) mm, rotated rx 0 ry 90 rz -60.43 deg; joints [19.527, -38.683, 128.45, -40.902, -89.823, 0.153]
  MoveL 549 to (514.85, 89.58, 0) mm, rotated rx 0 ry 90 rz -60.43 deg; joints [26.959, -33.163, 107.932, -34.418, -77.341, 8.54]
  MoveL 550 to (791.94, 89.58, 0) mm, rotated rx 0 ry 90 rz -60.43 deg; joints [22.642, -23.906, 83.37, -41.992, -66.325, 19.873]
  MoveL 551 to (893.34, 291.99, 0) mm, rotated rx 0 ry 90 rz -60.43 deg; joints [15.004, -22.457, 79.871, -50.3, -67.791, 24.48]
  Set speed (60.0 mm/s)
  MoveL 552 to (890.74, 291.64, 0) mm, rotated rx 0 ry 90 rz -60.43 deg; joints [15.038, -22.574, 80.152, -50.216, -67.881, 24.331]
  MoveL 553 to (888.19, 291.08, 0) mm, rotated rx 0 ry 90 rz -60.43 deg; joints [15.079, -22.686, 80.42, -50.127, -67.964, 24.187]
  MoveL 554 to (885.71, 290.29, 0) mm, rotated rx 0 ry 90 rz -60.43 deg; joints [15.127, -22.791, 80.673, -50.034, -68.04, 24.047]
  MoveL 555 to (883.3, 289.29, 0) mm, rotated rx 0 ry 90 rz -60.43 deg; joints [15.181, -22.89, 80.91, -49.938, -68.107, 23.913]
  MoveL 556 to (881, 288.07, 0) mm, rotated rx 0 ry 90 rz -60.43 deg; joints [15.241, -22.981, 81.128, -49.84, -68.165, 23.786]
  MoveL 557 to (878.81, 286.63, 0) mm, rotated rx 0 ry 90 rz -60.43 deg; joints [15.308, -23.063, 81.326, -49.739, -68.213, 23.666]
  MoveL 558 to (876.76, 284.98, 0) mm, rotated rx 0 ry 90 rz -60.43 deg; joints [15.38, -23.136, 81.502, -49.636, -68.25, 23.555]
  MoveL 559 to (874.88, 283.15, 0) mm, rotated rx 0 ry 90 rz -60.43 deg; joints [15.457, -23.198, 81.653, -49.533, -68.277, 23.455]
  MoveL 560 to (873.22, 281.16, 0) mm, rotated rx 0 ry 90 rz -60.43 deg; joints [15.538, -23.249, 81.775, -49.432, -68.291, 23.367]
  MoveL 561 to (871.77, 279.02, 0) mm, rotated rx 0 ry 90 rz -60.43 deg; joints [15.621, -23.287, 81.868, -49.333, -68.293, 23.292]
  MoveL 562 to (870.55, 276.75, 0) mm, rotated rx 0 ry 90 rz -60.43 deg; joints [15.707, -23.313, 81.931, -49.237, -68.284, 23.23]
  MoveL 563 to (869.59, 274.37, 0) mm, rotated rx 0 ry 90 rz -60.43 deg; joints [15.794, -23.327, 81.963, -49.145, -68.262, 23.183]
  MoveL 564 to (868.88, 271.89, 0) mm, rotated rx 0 ry 90 rz -60.43 deg; joints [15.882, -23.327, 81.964, -49.058, -68.227, 23.15]
  MoveL 565 to (868.44, 269.33, 0) mm, rotated rx 0 ry 90 rz -60.43 deg; joints [15.97, -23.314, 81.931, -48.977, -68.18, 23.133]
  MoveL 566 to (868.3, 266.7, 0) mm, rotated rx 0 ry 90 rz -60.43 deg; joints [16.057, -23.286, 81.865, -48.902, -68.121, 23.133]
  MoveL 567 to (868.3, 25.4, 0) mm, rotated rx 0 ry 90 rz -60.43 deg; joints [23.611, -19.084, 71.937, -43.202, -61.091, 24.418]
  MoveL 568 to (817.34, 25.4, 0) mm, rotated rx 0 ry 90 rz -60.43 deg; joints [24.292, -21.559, 77.733, -41.315, -63.283, 21.563]
  MoveL 569 to (817.34, 330.2, 0) mm, rotated rx 0 ry 90 rz -60.43 deg; joints [14.393, -26.193, 89.025, -49.367, -71.52, 20.274]
  MoveL 570 to (983.12, 330.2, 0) mm, rotated rx 0 ry 90 rz -60.43 deg; joints [13.065, -18.335, 70.208, -54.085, -65.279, 30.002]
  MoveL 571 to (1117.42, 127, 0) mm, rotated rx 0 ry 90 rz -60.43 deg; joints [17.967, -3.154, 36.898, -58.742, -52.161, 45.303]
  MoveL 572 to (1068.89, 127, 0) mm, rotated rx 0 ry 90 rz -60.43 deg; joints [18.415, -8.339, 47.974, -54.697, -55.097, 38.94]
  MoveL 573 to (967.85, 279.88, 0) mm, rotated rx 0 ry 90 rz -60.43 deg; joints [14.759, -18.492, 70.57, -52.381, -64.566, 29.131]
  MoveL 574 to (965.72, 282.67, 0) mm, rotated rx 0 ry 90 rz -60.43 deg; joints [14.689, -18.651, 70.936, -52.371, -64.726, 28.979]
  MoveL 575 to (963.26, 285.11, 0) mm, rotated rx 0 ry 90 rz -60.43 deg; joints [14.633, -18.821, 71.329, -52.342, -64.889, 28.807]
  MoveL 576 to (960.53, 287.21, 0) mm, rotated rx 0 ry 90 rz -60.43 deg; joints [14.59, -19.001, 71.743, -52.298, -65.054, 28.619]
  MoveL 577 to (957.55, 288.94, 0) mm, rotated rx 0 ry 90 rz -60.43 deg; joints [14.559, -19.186, 72.173, -52.237, -65.218, 28.419]
  MoveL 578 to (954.39, 290.31, 0) mm, rotated rx 0 ry 90 rz -60.43 deg; joints [14.542, -19.375, 72.612, -52.163, -65.379, 28.209]
  MoveL 579 to (951.08, 291.3, 0) mm, rotated rx 0 ry 90 rz -60.43 deg; joints [14.538, -19.566, 73.054, -52.077, -65.535, 27.992]
  MoveL 580 to (947.67, 291.9, 0) mm, rotated rx 0 ry 90 rz -60.43 deg; joints [14.547, -19.754, 73.493, -51.978, -65.685, 27.771]
  MoveL 581 to (944.2, 292.1, 0) mm, rotated rx 0 ry 90 rz -60.43 deg; joints [14.569, -19.939, 73.924, -51.87, -65.827, 27.55]
  MoveL 582 to (895.95, 292.1, 0) mm, rotated rx 0 ry 90 rz -60.43 deg; joints [14.978, -22.335, 79.58, -50.38, -67.693, 24.631]
  MoveL 583 to (893.34, 291.99, 0) mm, rotated rx 0 ry 90 rz -60.43 deg; joints [15.004, -22.457, 79.871, -50.3, -67.791, 24.48]
  MoveL 584 to (1117.81, 63.61, 0) mm, rotated rx 0 ry 90 rz -60.43 deg; joints [19.707, 0.123, 30.016, -59.745, -49.048, 48.333]
  Set speed (60.0 mm/s)
  MoveL 585 to (1115.19, 63.5, 0) mm, rotated rx 0 ry 90 rz -60.43 deg; joints [19.735, -0.316, 30.933, -59.364, -49.269, 47.772]
  MoveL 586 to (1066.94, 63.5, 0) mm, rotated rx 0 ry 90 rz -60.43 deg; joints [20.218, -6.4, 43.803, -54.303, -52.652, 40.176]
  MoveL 587 to (1060.06, 64.3, 0) mm, rotated rx 0 ry 90 rz -60.43 deg; joints [20.266, -7.108, 45.322, -53.759, -53.098, 39.324]
  MoveL 588 to (1056.75, 65.29, 0) mm, rotated rx 0 ry 90 rz -60.43 deg; joints [20.273, -7.459, 46.076, -53.51, -53.333, 38.915]
  MoveL 589 to (1053.59, 66.65, 0) mm, rotated rx 0 ry 90 rz -60.43 deg; joints [20.267, -7.801, 46.814, -53.28, -53.572, 38.523]
  MoveL 590 to (1050.62, 68.39, 0) mm, rotated rx 0 ry 90 rz -60.43 deg; joints [20.249, -8.132, 47.526, -53.072, -53.812, 38.153]
  MoveL 591 to (1047.88, 70.49, 0) mm, rotated rx 0 ry 90 rz -60.43 deg; joints [20.219, -8.446, 48.206, -52.89, -54.051, 37.81]
  MoveL 592 to (1045.42, 72.93, 0) mm, rotated rx 0 ry 90 rz -60.43 deg; joints [20.175, -8.742, 48.846, -52.734, -54.285, 37.496]
  MoveL 593 to (1043.29, 75.72, 0) mm, rotated rx 0 ry 90 rz -60.43 deg; joints [20.119, -9.015, 49.438, -52.608, -54.513, 37.217]
  MoveL 594 to (942.25, 228.6, 0) mm, rotated rx 0 ry 90 rz -60.43 deg; joints [16.582, -19.105, 71.984, -50.302, -64.2, 27.668]
  MoveL 595 to (893.72, 228.6, 0) mm, rotated rx 0 ry 90 rz -60.43 deg; joints [17.044, -21.572, 77.763, -48.68, -66.147, 24.701]
  MoveL 596 to (1028.02, 25.4, 0) mm, rotated rx 0 ry 90 rz -60.43 deg; joints [21.693, -8.674, 48.699, -51.28, -53.321, 36.688]
  MoveL 597 to (1193.8, 25.4, 0) mm, rotated rx 90 ry 70 rz 29.57 deg; joints [22.524, 4.177, 23.022, -59.584, -45.429, 30.087]
  MoveL 598 to (1193.8, 330.2, 0) mm, rotated rx 0 ry 90 rz -60.43 deg; joints [11.688, 0.316, 29.612, -66.361, -55.143, 52.555]
  MoveL 599 to (1142.85, 330.2, 0) mm, rotated rx 0 ry 90 rz -60.43 deg; joints [11.994, -6.514, 44.047, -61.62, -58.255, 44.243]
  MoveL 600 to (1142.85, 88.9, 0) mm, rotated rx 0 ry 90 rz -60.43 deg; joints [18.781, 3.597, 22.809, -63.431, -47.988, 53.233]
  MoveL 601 to (1142.7, 86.27, 0) mm, rotated rx 0 ry 90 rz -60.43 deg; joints [18.854, 3.808, 22.375, -63.553, -47.83, 53.463]
  MoveL 602 to (1142.26, 83.71, 0) mm, rotated rx 0 ry 90 rz -60.43 deg; joints [18.928, 3.936, 22.111, -63.604, -47.71, 53.588]
  MoveL 603 to (1141.56, 81.23, 0) mm, rotated rx 0 ry 90 rz -60.43 deg; joints [19.001, 3.978, 22.024, -63.582, -47.631, 53.602]
  MoveL 604 to (1140.59, 78.85, 0) mm, rotated rx 0 ry 90 rz -60.43 deg; joints [19.075, 3.935, 22.112, -63.486, -47.592, 53.508]
  MoveL 605 to (1139.37, 76.58, 0) mm, rotated rx 0 ry 90 rz -60.43 deg; joints [19.148, 3.811, 22.367, -63.32, -47.592, 53.309]
  MoveL 606 to (1137.93, 74.44, 0) mm, rotated rx 0 ry 90 rz -60.43 deg; joints [19.219, 3.613, 22.775, -63.09, -47.63, 53.016]
  MoveL 607 to (1136.26, 72.45, 0) mm, rotated rx 0 ry 90 rz -60.43 deg; joints [19.289, 3.35, 23.318, -62.806, -47.701, 52.641]
  MoveL 608 to (1134.38, 70.61, 0) mm, rotated rx 0 ry 90 rz -60.43 deg; joints [19.357, 3.032, 23.976, -62.477, -47.804, 52.196]
  MoveL 609 to (1132.33, 68.97, 0) mm, rotated rx 0 ry 90 rz -60.43 deg; joints [19.421, 2.67, 24.723, -62.115, -47.932, 51.7]
  MoveL 610 to (1130.15, 67.53, 0) mm, rotated rx 0 ry 90 rz -60.43 deg; joints [19.481, 2.279, 25.532, -61.733, -48.082, 51.17]
  MoveL 611 to (1127.84, 66.31, 0) mm, rotated rx 0 ry 90 rz -60.43 deg; joints [19.536, 1.867, 26.387, -61.338, -48.25, 50.617]
  MoveL 612 to (1125.43, 65.31, 0) mm, rotated rx 0 ry 90 rz -60.43 deg; joints [19.586, 1.44, 27.273, -60.937, -48.433, 50.05]
  MoveL 613 to (1122.95, 64.52, 0) mm, rotated rx 0 ry 90 rz -60.43 deg; joints [19.632, 1.004, 28.179, -60.535, -48.628, 49.476]
  MoveL 614 to (1120.4, 63.96, 0) mm, rotated rx 0 ry 90 rz -60.43 deg; joints [19.672, 0.564, 29.096, -60.137, -48.834, 48.903]
  MoveL 615 to (1117.81, 63.61, 0) mm, rotated rx 0 ry 90 rz -60.43 deg; joints [19.707, 0.123, 30.016, -59.745, -49.048, 48.333]
  MoveL 616 to (774.66, 25.4, 0) mm, rotated rx 0 ry 90 rz -60.43 deg; joints [24.891, -23.442, 82.242, -39.864, -65.068, 19.393]
  Set speed (60.0 mm/s)
  MoveL 617 to (464.73, 25.4, 0) mm, rotated rx 0 ry 90 rz -60.43 deg; joints [30.224, -33.544, 109.086, -31.013, -77.539, 7.391]
  MoveL 618 to (296.85, 279.4, 0) mm, rotated rx 0 ry 90 rz -60.43 deg; joints [23.416, -38.98, 130.17, -37.018, -90.95, -0.716]
  MoveL 619 to (345.39, 279.4, 0) mm, rotated rx 0 ry 90 rz -60.43 deg; joints [22.483, -38.373, 126.832, -37.956, -88.784, 0.948]
  MoveL 620 to (471.92, 87.94, 0) mm, rotated rx 0 ry 90 rz -60.43 deg; joints [27.828, -34.208, 111.146, -33.286, -79.024, 7.125]
  MoveL 621 to (476.14, 82.42, 0) mm, rotated rx 0 ry 90 rz -60.43 deg; joints [27.948, -34.037, 110.609, -33.204, -78.702, 7.306]
  MoveL 622 to (481.04, 77.53, 0) mm, rotated rx 0 ry 90 rz -60.43 deg; joints [28.032, -33.855, 110.043, -33.162, -78.37, 7.504]
  MoveL 623 to (486.53, 73.31, 0) mm, rotated rx 0 ry 90 rz -60.43 deg; joints [28.079, -33.665, 109.456, -33.16, -78.032, 7.716]
  MoveL 624 to (492.53, 69.8, 0) mm, rotated rx 0 ry 90 rz -60.43 deg; joints [28.09, -33.469, 108.857, -33.196, -77.693, 7.939]
  MoveL 625 to (498.88, 67.06, 0) mm, rotated rx 0 ry 90 rz -60.43 deg; joints [28.067, -33.271, 108.259, -33.268, -77.361, 8.169]
  MoveL 626 to (505.5, 65.09, 0) mm, rotated rx 0 ry 90 rz -60.43 deg; joints [28.011, -33.075, 107.668, -33.373, -77.04, 8.403]
  MoveL 627 to (519.21, 63.5, 0) mm, rotated rx 0 ry 90 rz -60.43 deg; joints [27.81, -32.695, 106.54, -33.675, -76.447, 8.875]
  MoveL 628 to (774.66, 63.5, 0) mm, rotated rx 0 ry 90 rz -60.43 deg; joints [23.7, -24.162, 83.994, -40.796, -66.248, 19.168]
  MoveL 629 to (774.66, 25.4, 0) mm, rotated rx 0 ry 90 rz -60.43 deg; joints [24.891, -23.442, 82.242, -39.864, -65.068, 19.393]
  MoveL 630 to (994.45, 406.4, 0) mm, rotated rx 0 ry 90 rz -60.43 deg; joints [10.582, -18.596, 70.808, -56.307, -66.727, 30.651]
  Set speed (60.0 mm/s)
  MoveL 631 to (1028.02, 355.6, 0) mm, rotated rx 0 ry 90 rz -60.43 deg; joints [11.963, -16.001, 64.886, -56.282, -64.15, 33.158]
  MoveL 632 to (1069.46, 355.6, 0) mm, rotated rx 0 ry 90 rz -60.43 deg; joints [11.698, -13.225, 58.671, -57.98, -62.434, 36.502]
  MoveL 633 to (1110.91, 355.6, 0) mm, rotated rx 0 ry 90 rz -60.43 deg; joints [11.444, -10.002, 51.584, -60.004, -60.601, 40.377]
  MoveL 634 to (1152.36, 355.6, 0) mm, rotated rx 0 ry 90 rz -60.43 deg; joints [11.201, -6.057, 43.069, -62.566, -58.569, 45.13]
  MoveL 635 to (1193.8, 355.6, 0) mm, rotated rx 0 ry 90 rz -60.43 deg; joints [10.968, -0.583, 31.49, -66.283, -56.105, 51.77]
  MoveL 636 to (1193.8, 431.8, 0) mm, rotated rx 0 ry 90 rz -60.43 deg; joints [8.786, -2.623, 35.776, -66.597, -58.698, 50.205]
  MoveL 637 to (1193.8, 508, 0) mm, rotated rx 0 ry 90 rz -60.43 deg; joints [6.578, -3.997, 38.681, -67.427, -60.983, 49.403]
  MoveL 638 to (1193.8, 584.2, 0) mm, rotated rx 0 ry 90 rz -60.43 deg; joints [4.351, -4.893, 40.585, -68.576, -63.048, 49.117]
  MoveL 639 to (1193.8, 660.4, 0) mm, rotated rx 0 ry 90 rz -60.43 deg; joints [2.11, -5.397, 41.659, -69.946, -64.946, 49.239]
  MoveL 640 to (1142.85, 660.4, 0) mm, rotated rx 0 ry 90 rz -60.43 deg; joints [2.166, -10.381, 52.41, -67.505, -67, 43.336]
  MoveL 641 to (1142.85, 419.1, 0) mm, rotated rx 0 ry 90 rz -60.43 deg; joints [9.394, -8.185, 47.642, -62.798, -60.952, 43.37]
  MoveL 642 to (1142.7, 416.47, 0) mm, rotated rx 0 ry 90 rz -60.43 deg; joints [9.472, -8.158, 47.583, -62.748, -60.884, 43.371]
  MoveL 643 to (1142.26, 413.91, 0) mm, rotated rx 0 ry 90 rz -60.43 deg; joints [9.55, -8.158, 47.584, -62.683, -60.831, 43.339]
  MoveL 644 to (1141.56, 411.43, 0) mm, rotated rx 0 ry 90 rz -60.43 deg; joints [9.626, -8.186, 47.643, -62.604, -60.793, 43.275]
  MoveL 645 to (1140.59, 409.05, 0) mm, rotated rx 0 ry 90 rz -60.43 deg; joints [9.701, -8.239, 47.758, -62.51, -60.77, 43.182]
  MoveL 646 to (1139.37, 406.78, 0) mm, rotated rx 0 ry 90 rz -60.43 deg; joints [9.774, -8.317, 47.926, -62.405, -60.762, 43.06]
  MoveL 647 to (1137.93, 404.64, 0) mm, rotated rx 0 ry 90 rz -60.43 deg; joints [9.845, -8.418, 48.145, -62.287, -60.768, 42.912]
  MoveL 648 to (1136.26, 402.65, 0) mm, rotated rx 0 ry 90 rz -60.43 deg; joints [9.912, -8.541, 48.41, -62.16, -60.789, 42.74]
  MoveL 649 to (1134.38, 400.81, 0) mm, rotated rx 0 ry 90 rz -60.43 deg; joints [9.976, -8.684, 48.721, -62.024, -60.824, 42.544]
  MoveL 650 to (1132.33, 399.17, 0) mm, rotated rx 0 ry 90 rz -60.43 deg; joints [10.035, -8.845, 49.07, -61.881, -60.872, 42.33]
  MoveL 651 to (1130.15, 397.73, 0) mm, rotated rx 0 ry 90 rz -60.43 deg; joints [10.089, -9.02, 49.45, -61.735, -60.933, 42.101]
  MoveL 652 to (1127.84, 396.51, 0) mm, rotated rx 0 ry 90 rz -60.43 deg; joints [10.138, -9.207, 49.856, -61.587, -61.005, 41.861]
  MoveL 653 to (1125.43, 395.51, 0) mm, rotated rx 0 ry 90 rz -60.43 deg; joints [10.18, -9.405, 50.284, -61.438, -61.086, 41.611]
  MoveL 654 to (1122.95, 394.72, 0) mm, rotated rx 0 ry 90 rz -60.43 deg; joints [10.217, -9.61, 50.731, -61.29, -61.178, 41.354]
  MoveL 655 to (1120.4, 394.15, 0) mm, rotated rx 0 ry 90 rz -60.43 deg; joints [10.247, -9.822, 51.192, -61.144, -61.278, 41.093]
  MoveL 656 to (1117.81, 393.81, 0) mm, rotated rx 0 ry 90 rz -60.43 deg; joints [10.271, -10.039, 51.664, -61.001, -61.386, 40.828]
  MoveL 657 to (1115.19, 393.7, 0) mm, rotated rx 0 ry 90 rz -60.43 deg; joints [10.289, -10.258, 52.143, -60.863, -61.5, 40.563]
  MoveL 658 to (1066.94, 393.7, 0) mm, rotated rx 0 ry 90 rz -60.43 deg; joints [10.556, -13.932, 60.244, -58.637, -63.565, 36.144]
  MoveL 659 to (1063.47, 393.9, 0) mm, rotated rx 0 ry 90 rz -60.43 deg; joints [10.57, -14.174, 60.784, -58.499, -63.713, 35.854]
  MoveL 660 to (1060.06, 394.5, 0) mm, rotated rx 0 ry 90 rz -60.43 deg; joints [10.571, -14.415, 61.322, -58.373, -63.868, 35.572]
  MoveL 661 to (1056.75, 395.49, 0) mm, rotated rx 0 ry 90 rz -60.43 deg; joints [10.56, -14.651, 61.85, -58.262, -64.028, 35.3]
  MoveL 662 to (1053.59, 396.85, 0) mm, rotated rx 0 ry 90 rz -60.43 deg; joints [10.536, -14.879, 62.361, -58.167, -64.191, 35.041]
  MoveL 663 to (1050.62, 398.59, 0) mm, rotated rx 0 ry 90 rz -60.43 deg; joints [10.499, -15.097, 62.85, -58.089, -64.355, 34.8]
  MoveL 664 to (1047.88, 400.69, 0) mm, rotated rx 0 ry 90 rz -60.43 deg; joints [10.45, -15.301, 63.31, -58.03, -64.518, 34.579]
  MoveL 665 to (1045.42, 403.13, 0) mm, rotated rx 0 ry 90 rz -60.43 deg; joints [10.389, -15.49, 63.734, -57.991, -64.677, 34.382]
  MoveL 666 to (1043.29, 405.92, 0) mm, rotated rx 0 ry 90 rz -60.43 deg; joints [10.314, -15.66, 64.117, -57.974, -64.832, 34.211]
  MoveL 667 to (942.25, 558.8, 0) mm, rotated rx 0 ry 90 rz -60.43 deg; joints [5.848, -22.466, 79.892, -59.065, -71.819, 27.503]
  MoveL 668 to (893.72, 558.8, 0) mm, rotated rx 0 ry 90 rz -60.43 deg; joints [6.02, -24.703, 85.32, -58.051, -73.408, 24.603]
  MoveL 669 to (927.3, 508, 0) mm, rotated rx 0 ry 90 rz -60.43 deg; joints [7.613, -22.894, 80.92, -57.237, -71.335, 26.442]
  MoveL 670 to (960.87, 457.2, 0) mm, rotated rx 0 ry 90 rz -60.43 deg; joints [9.133, -20.872, 76.111, -56.644, -69.113, 28.44]
  MoveL 671 to (994.45, 406.4, 0) mm, rotated rx 0 ry 90 rz -60.43 deg; joints [10.582, -18.596, 70.808, -56.307, -66.727, 30.651]
  Set speed (2000.0 mm/s)
  MoveL 672 to (994.45, 406.4, 0) mm, rotated rx 0 ry 90 rz -60.43 deg; joints [10.582, -18.596, 70.808, -56.307, -66.727, 30.651]
  MoveL 673 to (994.45, 406.4, 10) mm, rotated rx 0 ry 90 rz -60.43 deg; joints [10.582, -19.112, 71.071, -56.398, -66.586, 30.882]

--- program Prog2 (robot KUKA KR 30 HA) ---
  MoveC [its target is no longer in the station] [its target is no longer in the station]
